# B&R Automation Studio project DiCoS_ACOPOStrak
Automation Studio 4.12.2.93; technology packages: mapp 5.21.0, mappCockpit 5.21.0, mappMotion 5.21.2, mappView 5.21.0

## Configuration Config2

CPU 5PC900.TS17-00, AutomationRuntime C4.90, Build 4.1.2, Safety 0.0, Vc V4.72.2

### Task classes (Cpu.sw)
```
Cyclic#1 (cycle 800 us, tolerance 0 us):
  trakFSM <- TrakControl.trakFSM.prg
  trakMove <- TrakControl.trakMove.prg
DataObjects: McAcpSys
Binaries: FWRules, McAcpSim, arcoal, arsvcreg, TCData, McAcpDrv, arflatprv, udbdef, McProfGen, mvLoader, mCoWebSc, asnxdb1, ConfAsmb, ConfSec, ConfShut, iomap, arconfig, asfw, ashwac, sysconf, User, Role, ashwd, Settings, Config_1, ConfPP, ConfCoup
Libraries: McBase, McAxis, McAcpTrak, AsIORTI, AsBrStr, McPureVAx, CoTrace, AsZip, FileIO, runtime, MpAxis, MpBase, McAcpAx, powerlnk, asieccon, arssl, asepl, MpData, sys_lib, DataObj, brsystem, astime
```

### Hardware
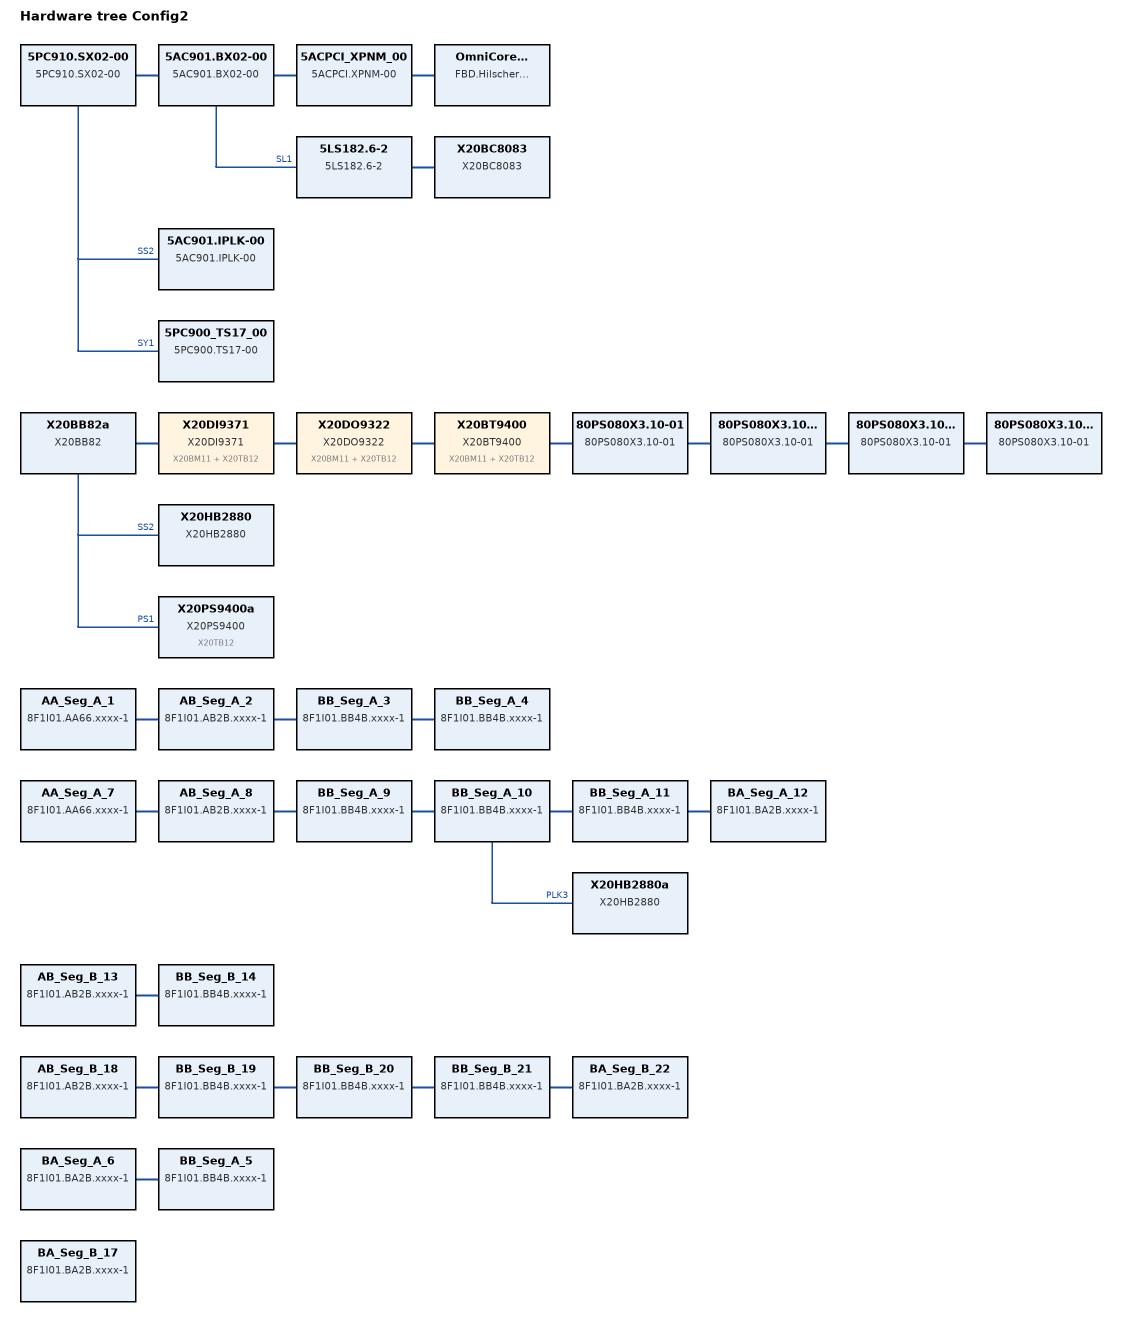
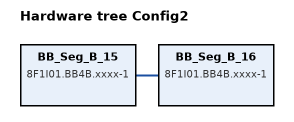
```
5AC901.BX02-00 : 5AC901.BX02-00 v1.0.1.0  [SY -> 5PC910.SX02-00.SY3]
5AC901.IPLK-00 : 5AC901.IPLK-00 v1.8.0.1  [SS -> 5PC910.SX02-00.SS2]
  Connector IF1:
    DNAConfiguration = manual
    EplNatSubnet = 192.168.102.0
5ACPCI_XPNM_00 : 5ACPCI.XPNM-00 v1.3.1.0  [SL -> 5AC901.BX02-00.SL2]
  Connector IF1:
    DtmId = d6364a6a-af48-4c58-9fae-63d24b23d839
  ConfigFile = 5ACPCI_XPNM_00.dtm
  ConfigModule = asnxdb1
5LS182.6-2 : 5LS182.6-2 v1.9.0.0  [SL -> 5AC901.BX02-00.SL1]
  Connector IF1:
    MtuSize = 1500
    CycleTime = 800
    EplNatSubnet = 192.168.103.0
5PC900_TS17_00 : 5PC900.TS17-00 v2.1.0.0  [SY -> 5PC910.SX02-00.SY1]
  ConfigurationID = APT_BFH_HW_Config
  TimerDeviceType = EPLX2X
  TimerDevice = 5LS182.6-2.IF1
  TaskClassIdleTime = 1600
  Cyclic1Duration = 800
  Cyclic1Tolerance = 0
  Cyclic3Duration = 49600
  Cyclic3Tolerance = 49600
  Cyclic8Duration = 9600
  FileDevice1
  FileDeviceName1 = SvgData
  FileDevicePath1 = C:\Users\nikla\Documents\BrAutomation\DiCoS_ACOPOStrak\Trak
  FileDevice2
  FileDeviceName2 = User
  FileDevicePath2 = C:\Users\nikla\Documents\BrAutomation\DiCoS_ACOPOStrak\Trak\User
  ActivateOpcUa = 1
  OpcUa_AuthenticationSecurityPolicy_EnableNone = 1
  OpcUa_AuthenticationSecurityPolicy_EnableBasic128Rsa15 = 1
  OpcUaInformationModels_PV_Version = 1
5PC910.SX02-00 : 5PC910.SX02-00 v2.1.0.0
  Connector IF1:
    AssignedOperatingSystem = ARemb
  Connector IF3:
    AssignedOperatingSystem = ARemb
    ActivateDevice = 1
    Mode = Manual
    InternetAddress = 192.168.1.220
    SubnetMask = 255.255.255.0
  Connector IF4:
    AssignedOperatingSystem = ARemb
    ActivateDevice = 1
    Mode = Manual
    InternetAddress = 10.0.0.3
    SubnetMask = 255.255.255.0
    ActivateSnmp = 2
  Connector IF5:
    AssignedOperatingSystem = ARemb
  Connector IF6:
    AssignedOperatingSystem = ARemb
  Connector IF7:
    AssignedOperatingSystem = ARemb
  Connector IF8:
    AssignedOperatingSystem = ARemb
  Connector IF9:
    AssignedOperatingSystem = ARemb
80PS080X3.10-01 : 80PS080X3.10-01 v1.5.0.0  [X2X1 -> X20BT9400.X2X1 [Cable Type=X2XCable, Length=10, Version=1.0.0.3]]
  Supervision = off
  ParallelMode01 = on
  VoltageSet01 = 58
  RampMode01 = steep
  ChopperEnable01 = on
80PS080X3.10-01a : 80PS080X3.10-01 v1.5.0.0  [X2X1 -> 80PS080X3.10-01.X2X2 [Cable Type=X2XCable, Length=10, Version=1.0.0.3]]
  Supervision = off
  ParallelMode01 = on
  VoltageSet01 = 58
  RampMode01 = steep
  ChopperEnable01 = on
80PS080X3.10-01b : 80PS080X3.10-01 v1.5.0.0  [X2X1 -> 80PS080X3.10-01a.X2X2 [Cable Type=X2XCable, Length=10, Version=1.0.0.3]]
  Supervision = off
  ParallelMode01 = on
  VoltageSet01 = 58
  RampMode01 = steep
  ChopperEnable01 = on
80PS080X3.10-01c : 80PS080X3.10-01 v1.5.0.0  [X2X1 -> 80PS080X3.10-01b.X2X2 [Cable Type=X2XCable, Length=10, Version=1.0.0.3]]
  Supervision = off
  ParallelMode01 = on
  VoltageSet01 = 58
  RampMode01 = steep
  ChopperEnable01 = on
AA_Seg_A_1 : 8F1I01.AA66.xxxx-1 v1.0.0.2  [PLK1 -> BA_Seg_A_12.PLK2 (NodeNumber=1) [Cable Type=PowerlinkCable, Length=10, Version=1.0.0.3]; PLK2 -> AB_Seg_A_2.PLK1 (NodeNumber=1) [Cable Type=PowerlinkCable, Length=10, Version=1.0.0.3]]
  EnableDNA = on
  DriveConfiguration:
    McTypeID = LLMConfig
  DriveConfiguration/Segment:
    Shape = STRAIGHT660
    SegmentReference = Seg_A_1
    StopReaction = UseAssemblySetting
    SpeedFilter = UseAssemblySetting
AA_Seg_A_7 : 8F1I01.AA66.xxxx-1 v1.0.0.2  [PLK1 -> BA_Seg_A_6.PLK2 (NodeNumber=7) [Cable Type=PowerlinkCable, Length=10, Version=1.0.0.3]; PLK2 -> AB_Seg_A_8.PLK1 (NodeNumber=7) [Cable Type=PowerlinkCable, Length=10, Version=1.0.0.3]]
  EnableDNA = on
  DriveConfiguration:
    McTypeID = LLMConfig
  DriveConfiguration/Segment:
    Shape = STRAIGHT660
    SegmentReference = Seg_A_7
    SegmentSectorDirection = Positive
    ElongationCompensation = UseAssemblySetting
    StopReaction = UseAssemblySetting
    SpeedFilter = UseAssemblySetting
AB_Seg_A_2 : 8F1I01.AB2B.xxxx-1 v1.0.0.2  [PLK1 -> AA_Seg_A_1.PLK2 (NodeNumber=2) [Cable Type=PowerlinkCable, Length=10, Version=1.0.0.3]; PLK2 -> BB_Seg_A_3.PLK1 (NodeNumber=2) [Cable Type=PowerlinkCable, Length=10, Version=1.0.0.3]]
  EnableDNA = on
  DriveConfiguration:
    McTypeID = LLMConfig
  DriveConfiguration/Segment:
    Shape = STRAIGHT105_TO_CIRCULAR
    SegmentReference = Seg_A_2
    StopReaction = UseAssemblySetting
    SpeedFilter = UseAssemblySetting
AB_Seg_A_8 : 8F1I01.AB2B.xxxx-1 v1.0.0.2  [PLK1 -> AA_Seg_A_7.PLK2 (NodeNumber=8) [Cable Type=PowerlinkCable, Length=10, Version=1.0.0.3]; PLK2 -> BB_Seg_A_9.PLK1 (NodeNumber=8) [Cable Type=PowerlinkCable, Length=10, Version=1.0.0.3]]
  EnableDNA = on
  DriveConfiguration:
    McTypeID = LLMConfig
  DriveConfiguration/Segment:
    Shape = STRAIGHT105_TO_CIRCULAR
    SegmentReference = Seg_A_8
    StopReaction = UseAssemblySetting
    SpeedFilter = UseAssemblySetting
AB_Seg_B_13 : 8F1I01.AB2B.xxxx-1 v1.0.0.2  [PLK1 -> BA_Seg_B_22.PLK2 (NodeNumber=13) [Cable Type=PowerlinkCable, Length=10, Version=1.0.0.3]; PLK2 -> BB_Seg_B_14.PLK1 (NodeNumber=13) [Cable Type=PowerlinkCable, Length=10, Version=1.0.0.3]]
  EnableDNA = on
  DriveConfiguration:
    McTypeID = LLMConfig
  DriveConfiguration/Segment:
    Shape = STRAIGHT105_TO_CIRCULAR
    SegmentReference = Seg_B_13
    StopReaction = UseAssemblySetting
    SpeedFilter = UseAssemblySetting
AB_Seg_B_18 : 8F1I01.AB2B.xxxx-1 v1.0.0.2  [PLK1 -> BA_Seg_B_17.PLK2 (NodeNumber=18) [Cable Type=PowerlinkCable, Length=10, Version=1.0.0.3]; PLK2 -> BB_Seg_B_19.PLK1 (NodeNumber=18) [Cable Type=PowerlinkCable, Length=10, Version=1.0.0.3]]
  EnableDNA = on
  DriveConfiguration:
    McTypeID = LLMConfig
  DriveConfiguration/Segment:
    Shape = STRAIGHT105_TO_CIRCULAR
    SegmentReference = Seg_B_18
    StopReaction = UseAssemblySetting
    SpeedFilter = UseAssemblySetting
BA_Seg_A_12 : 8F1I01.BA2B.xxxx-1 v1.0.0.2  [PLK1 -> BB_Seg_A_11.PLK2 (NodeNumber=12) [Cable Type=PowerlinkCable, Length=10, Version=1.0.0.3]; PLK2 -> AA_Seg_A_1.PLK1 (NodeNumber=12) [Cable Type=PowerlinkCable, Length=10, Version=1.0.0.3]]
  EnableDNA = on
  DriveConfiguration:
    McTypeID = LLMConfig
  DriveConfiguration/Segment:
    Shape = CIRCULAR_TO_STRAIGHT105
    SegmentReference = Seg_A_12
    StopReaction = UseAssemblySetting
    SpeedFilter = UseAssemblySetting
BA_Seg_A_6 : 8F1I01.BA2B.xxxx-1 v1.0.0.2  [PLK1 -> BB_Seg_A_5.PLK2 (NodeNumber=6) [Cable Type=PowerlinkCable, Length=10, Version=1.0.0.3]; PLK2 -> AA_Seg_A_7.PLK1 (NodeNumber=6) [Cable Type=PowerlinkCable, Length=10, Version=1.0.0.3]]
  EnableDNA = on
  DriveConfiguration:
    McTypeID = LLMConfig
  DriveConfiguration/Segment:
    Shape = CIRCULAR_TO_STRAIGHT105
    SegmentReference = Seg_A_6
    StopReaction = UseAssemblySetting
    SpeedFilter = UseAssemblySetting
BA_Seg_B_17 : 8F1I01.BA2B.xxxx-1 v1.0.0.2  [PLK1 -> BB_Seg_B_16.PLK2 (NodeNumber=17) [Cable Type=PowerlinkCable, Length=10, Version=1.0.0.3]; PLK2 -> AB_Seg_B_18.PLK1 (NodeNumber=17) [Cable Type=PowerlinkCable, Length=10, Version=1.0.0.3]]
  EnableDNA = on
  DriveConfiguration:
    McTypeID = LLMConfig
  DriveConfiguration/Segment:
    Shape = CIRCULAR_TO_STRAIGHT105
    SegmentReference = Seg_B_17
    StopReaction = UseAssemblySetting
    SpeedFilter = UseAssemblySetting
BA_Seg_B_22 : 8F1I01.BA2B.xxxx-1 v1.0.0.2  [PLK1 -> BB_Seg_B_21.PLK2 (NodeNumber=22) [Cable Type=PowerlinkCable, Length=10, Version=1.0.0.3]; PLK2 -> AB_Seg_B_13.PLK1 (NodeNumber=22) [Cable Type=PowerlinkCable, Length=10, Version=1.0.0.3]]
  EnableDNA = on
  DriveConfiguration:
    McTypeID = LLMConfig
  DriveConfiguration/Segment:
    Shape = CIRCULAR_TO_STRAIGHT105
    SegmentReference = Seg_B_22
    StopReaction = UseAssemblySetting
    SpeedFilter = UseAssemblySetting
BB_Seg_A_10 : 8F1I01.BB4B.xxxx-1 v1.0.0.2  [PLK1 -> BB_Seg_A_9.PLK2 (NodeNumber=10) [Cable Type=PowerlinkCable, Length=10, Version=1.0.0.3]; PLK2 -> BB_Seg_A_11.PLK1 (NodeNumber=10) [Cable Type=PowerlinkCable, Length=10, Version=1.0.0.3]; PLK3 -> X20HB2880a.ETH1 (NodeNumber=10) [Cable Type=PowerlinkCable, Length=10, Version=1.0.0.3]]
  EnableDNA = on
  DriveConfiguration:
    McTypeID = LLMConfig
  DriveConfiguration/Segment:
    Shape = CIRCULAR
    SegmentReference = Seg_A_10
    StopReaction = UseAssemblySetting
    SpeedFilter = UseAssemblySetting
BB_Seg_A_11 : 8F1I01.BB4B.xxxx-1 v1.0.0.2  [PLK1 -> BB_Seg_A_10.PLK2 (NodeNumber=11) [Cable Type=PowerlinkCable, Length=10, Version=1.0.0.3]; PLK2 -> BA_Seg_A_12.PLK1 (NodeNumber=11) [Cable Type=PowerlinkCable, Length=10, Version=1.0.0.3]]
  EnableDNA = on
  DriveConfiguration:
    McTypeID = LLMConfig
  DriveConfiguration/Segment:
    Shape = CIRCULAR
    SegmentReference = Seg_A_11
    StopReaction = UseAssemblySetting
    SpeedFilter = UseAssemblySetting
BB_Seg_A_3 : 8F1I01.BB4B.xxxx-1 v1.0.0.2  [PLK1 -> AB_Seg_A_2.PLK2 (NodeNumber=3) [Cable Type=PowerlinkCable, Length=10, Version=1.0.0.3]; PLK2 -> BB_Seg_A_4.PLK1 (NodeNumber=3) [Cable Type=PowerlinkCable, Length=10, Version=1.0.0.3]]
  EnableDNA = on
  DriveConfiguration:
    McTypeID = LLMConfig
  DriveConfiguration/Segment:
    Shape = CIRCULAR
    SegmentReference = Seg_A_3
    StopReaction = UseAssemblySetting
    SpeedFilter = UseAssemblySetting
BB_Seg_A_4 : 8F1I01.BB4B.xxxx-1 v1.0.0.2  [PLK1 -> BB_Seg_A_3.PLK2 (NodeNumber=4) [Cable Type=PowerlinkCable, Length=10, Version=1.0.0.3]]
  EnableDNA = on
  DriveConfiguration:
    McTypeID = LLMConfig
  DriveConfiguration/Segment:
    Shape = CIRCULAR
    SegmentReference = Seg_A_4
    StopReaction = UseAssemblySetting
    SpeedFilter = UseAssemblySetting
BB_Seg_A_5 : 8F1I01.BB4B.xxxx-1 v1.0.0.2  [PLK2 -> BA_Seg_A_6.PLK1 (NodeNumber=5) [Cable Type=PowerlinkCable, Length=10, Version=1.0.0.3]]
  EnableDNA = on
  DriveConfiguration:
    McTypeID = LLMConfig
  DriveConfiguration/Segment:
    Shape = CIRCULAR
    SegmentReference = Seg_A_5
    StopReaction = UseAssemblySetting
    SpeedFilter = UseAssemblySetting
BB_Seg_A_9 : 8F1I01.BB4B.xxxx-1 v1.0.0.2  [PLK1 -> AB_Seg_A_8.PLK2 (NodeNumber=9) [Cable Type=PowerlinkCable, Length=10, Version=1.0.0.3]; PLK2 -> BB_Seg_A_10.PLK1 (NodeNumber=9) [Cable Type=PowerlinkCable, Length=10, Version=1.0.0.3]]
  EnableDNA = on
  DriveConfiguration:
    McTypeID = LLMConfig
  DriveConfiguration/Segment:
    Shape = CIRCULAR
    SegmentReference = Seg_A_9
    StopReaction = UseAssemblySetting
    SpeedFilter = UseAssemblySetting
BB_Seg_B_14 : 8F1I01.BB4B.xxxx-1 v1.0.0.2  [PLK1 -> AB_Seg_B_13.PLK2 (NodeNumber=14) [Cable Type=PowerlinkCable, Length=10, Version=1.0.0.3]]
  EnableDNA = on
  DriveConfiguration:
    McTypeID = LLMConfig
  DriveConfiguration/Segment:
    Shape = CIRCULAR
    SegmentReference = Seg_B_14
    StopReaction = UseAssemblySetting
    SpeedFilter = UseAssemblySetting
BB_Seg_B_15 : 8F1I01.BB4B.xxxx-1 v1.0.0.2  [PLK2 -> BB_Seg_B_16.PLK1 (NodeNumber=15) [Cable Type=PowerlinkCable, Length=10, Version=1.0.0.3]]
  EnableDNA = on
  DriveConfiguration:
    McTypeID = LLMConfig
  DriveConfiguration/Segment:
    Shape = CIRCULAR
    SegmentReference = Seg_B_15
    StopReaction = UseAssemblySetting
    SpeedFilter = UseAssemblySetting
BB_Seg_B_16 : 8F1I01.BB4B.xxxx-1 v1.0.0.2  [PLK1 -> BB_Seg_B_15.PLK2 (NodeNumber=16) [Cable Type=PowerlinkCable, Length=10, Version=1.0.0.3]; PLK2 -> BA_Seg_B_17.PLK1 (NodeNumber=16) [Cable Type=PowerlinkCable, Length=10, Version=1.0.0.3]]
  EnableDNA = on
  DriveConfiguration:
    McTypeID = LLMConfig
  DriveConfiguration/Segment:
    Shape = CIRCULAR
    SegmentReference = Seg_B_16
    StopReaction = UseAssemblySetting
    SpeedFilter = UseAssemblySetting
BB_Seg_B_19 : 8F1I01.BB4B.xxxx-1 v1.0.0.2  [PLK1 -> AB_Seg_B_18.PLK2 (NodeNumber=19) [Cable Type=PowerlinkCable, Length=10, Version=1.0.0.3]; PLK2 -> BB_Seg_B_20.PLK1 (NodeNumber=19) [Cable Type=PowerlinkCable, Length=10, Version=1.0.0.3]]
  EnableDNA = on
  DriveConfiguration:
    McTypeID = LLMConfig
  DriveConfiguration/Segment:
    Shape = CIRCULAR
    SegmentReference = Seg_B_19
    StopReaction = UseAssemblySetting
    SpeedFilter = UseAssemblySetting
BB_Seg_B_20 : 8F1I01.BB4B.xxxx-1 v1.0.0.2  [PLK1 -> BB_Seg_B_19.PLK2 (NodeNumber=20) [Cable Type=PowerlinkCable, Length=10, Version=1.0.0.3]; PLK2 -> BB_Seg_B_21.PLK1 (NodeNumber=20) [Cable Type=PowerlinkCable, Length=10, Version=1.0.0.3]; PLK3 -> X20HB2880a.ETH2 (NodeNumber=20) [Cable Type=PowerlinkCable, Length=10, Version=1.0.0.3]]
  EnableDNA = on
  DriveConfiguration:
    McTypeID = LLMConfig
  DriveConfiguration/Segment:
    Shape = CIRCULAR
    SegmentReference = Seg_B_20
    StopReaction = UseAssemblySetting
    SpeedFilter = UseAssemblySetting
BB_Seg_B_21 : 8F1I01.BB4B.xxxx-1 v1.0.0.2  [PLK1 -> BB_Seg_B_20.PLK2 (NodeNumber=21) [Cable Type=PowerlinkCable, Length=10, Version=1.0.0.3]; PLK2 -> BA_Seg_B_22.PLK1 (NodeNumber=21) [Cable Type=PowerlinkCable, Length=10, Version=1.0.0.3]]
  EnableDNA = on
  DriveConfiguration:
    McTypeID = LLMConfig
  DriveConfiguration/Segment:
    Shape = CIRCULAR
    SegmentReference = Seg_B_21
    StopReaction = UseAssemblySetting
    SpeedFilter = UseAssemblySetting
OmniCore_Standard : FBD.Hilscher.PNIOGenDevDTM2.OmniCore Standard v1.1 (OrderNumber=OmniCore Standard, VendorAddress=omnicore)  [PN1 -> 5ACPCI_XPNM_00.IF1]
  DtmId = 5f4a343d-d0a2-4fff-bfd8-5abcfec9ae3d
X20BB82a : X20BB82 v1.1.0.0
  Connector IF1:
    CycleTime = 1600
X20BC8083 : X20BC8083 v2.14.0.0  [PLK1 -> 5LS182.6-2.IF1 (NodeNumber=23) [Cable Type=PowerlinkCable, Length=10, Version=1.0.0.3]; SL -> X20BB82a.SL1]
  Supervision = off
  EPL_Chained = on
  EnableDNA = on
X20BM11 : X20BM11 v1.1.0.0  [X2X1 -> X20BM11b.X2X2]
X20BM11a : X20BM11 v1.1.0.0  [X2X1 -> X20BB82a.IF1]
X20BM11b : X20BM11 v1.1.0.0  [X2X1 -> X20BM11a.X2X2]
X20BT9400 : X20BT9400 v1.3.0.0  [SS1 -> X20TB12.SS; SL -> X20BM11.SL1]
  Supervision = off
X20DI9371 : X20DI9371 v1.4.0.0  [SS1 -> X20TB12b.SS; SL -> X20BM11a.SL1]
X20DO9322 : X20DO9322 v1.5.0.0  [SS1 -> X20TB12c.SS; SL -> X20BM11b.SL1]
X20HB2880 : X20HB2880 v1.2.0.0  [SS -> X20BB82a.SS2]
X20HB2880a : X20HB2880 v1.2.0.0  [ETH1 -> BB_Seg_A_10.PLK3 [Cable Type=PowerlinkCable, Length=10, Version=1.0.0.3]; ETH2 -> BB_Seg_B_20.PLK3 [Cable Type=PowerlinkCable, Length=10, Version=1.0.0.3]; SS -> X20BB82a.SS1]
X20PS9400a : X20PS9400 v1.8.0.0  [SS1 -> X20TB12a.SS; PS -> X20BB82a.PS1]
X20TB12 : X20TB12 v1.0.0.0
X20TB12a : X20TB12 v1.0.0.0
X20TB12b : X20TB12 v1.0.0.0
X20TB12c : X20TB12 v1.0.0.0
```

### ConfAsmb.assembly - 5PC900_TS17_00/mappMotion/ConfAsmb.assembly
```
Element gAssemblyFigure8 (Type=assembly)
  Tracks:
    TrackSeparation = 0.030
    Track[1]:
      Segments:
        SegmentRef[1] = ::Seg_A_1
        SegmentRef[2] = ::Seg_A_2
        SegmentRef[3] = ::Seg_A_3
        SegmentRef[4] = ::Seg_A_4
        SegmentRef[5] = ::Seg_A_5
        SegmentRef[6] = ::Seg_A_6
        SegmentRef[7] = ::Seg_A_7
        SegmentRef[8] = ::Seg_A_8
        SegmentRef[9] = ::Seg_A_9
        SegmentRef[10] = ::Seg_A_10
        SegmentRef[11] = ::Seg_A_11
        SegmentRef[12] = ::Seg_A_12
      Position = Absolute
        SegmentRef = ::Seg_A_1
        SegmentCountDirection = RightToLeft
        Translation:
          X = 0.0
          Y = 0.0
          Z = 0.0
        Orientation:
          Angle1 = 0.0
          Angle2 = 0.0
          Angle3 = 180.0
    Track[2]:
      Segments:
        SegmentRef[1] = ::Seg_B_13
        SegmentRef[2] = ::Seg_B_14
        SegmentRef[3] = ::Seg_B_15
        SegmentRef[4] = ::Seg_B_16
        SegmentRef[5] = ::Seg_B_17
        SegmentRef[6] = ::Seg_B_18
        SegmentRef[7] = ::Seg_B_19
        SegmentRef[8] = ::Seg_B_20
        SegmentRef[9] = ::Seg_B_21
        SegmentRef[10] = ::Seg_B_22
      Position = RelativeToOne
        TrackSegmentPosition:
          SegmentRef = ::Seg_B_13
        Base:
          SegmentRef = ::Seg_A_7
          Position = 0.329907
  CommonSegmentSettings:
    SegmentSimulationOnPLC = Off
    ElongationCompensation = Inactive
    StopReaction = InductionHalt
    SpeedFilter = Lowpass
      FilterTime = 0.0008
    ControllerParameters:
      DefaultParameter:
        Controller:
          Position:
            ProportionalGain = 150
          Speed:
            ProportionalGain = 80
            IntegrationTime = 0
          FeedForward:
            TotalMass = 0.7
            ForcePositive = 1.5
            ForceNegative = 1.5
            SpeedForceFactor = 1.4
            ForceLoad = 0.0
        MovementErrorLimits:
          PositionError = 0.03
          VelocityError = 50
      AdditionalParameterSets = NotUsed
    ScopeOfErrorReaction = Assembly
    ShuttleIdentificationTime = 0
  Shuttles:
    MaxShuttleCount = 10
    MaxShuttleCommandCount = 0
    UseConvoys = Active
    DistanceReserve:
      Collision = 0.002
      ErrorStop = 0.006
    ShuttleStereotypes:
      ShuttleStRef[1] = gShuttleStereotype_1
    MagnetPlateConfigurations:
      ShuttleType[1] = 8F1SA.100.xxxxxx-x
    CollisionAvoidance:
      Strategy = Constant
      MaximumModelDimensions:
        Length:
          ExtentToFront = 0.046
          ExtentToBack = 0.046
        Width:
          Width = 0.046
  AssemblyFeatures:
    AssemblyFeatureRef[1] = Feature_Coupling
  Visualization:
    MonitoringPv = ::trakAsmb.monData
    ProcessingTaskClass = 1
```

### ConfCoup.assemblyfeature - 5PC900_TS17_00/mappMotion/ConfCoup.assemblyfeature
```
Element Feature_Coupling (Type=assemblyfeature)
  Type = Coupling
    CouplingObject[1]:
      Name = couplingLoad
      ShuttleCount = 1
      CamAutomat
      CamList
```

### ConfPP.processpointlist - 5PC900_TS17_00/mappMotion/ConfPP.processpointlist
```
Element gPPList (Type=processpointlist)
  ProcessPoint[0]:
    Name = gPPDepot
    SectorRef = gSecFull
    Position = 5.6
    TriggerEventBufferSize = 10
    BarrierFunctionality = On
```

### ConfSec.sector - 5PC900_TS17_00/mappMotion/ConfSec.sector
```
Element gSecMajor (Type=sector)
  Type = Composed
    StartSegment:
      SegmentRef = ::Seg_A_3
    IntermediateSegments:
      SegmentRef[1] = ::Seg_A_2
      SegmentRef[2] = ::Seg_A_1
      SegmentRef[3] = ::Seg_A_12
      SegmentRef[4] = ::Seg_A_11
      SegmentRef[5] = ::Seg_A_10
      SegmentRef[6] = ::Seg_A_9
      SegmentRef[7] = ::Seg_A_8
      SegmentRef[8] = ::Seg_A_7
      SegmentRef[9] = ::Seg_A_6
      SegmentRef[10] = ::Seg_A_5
    EndSegment:
      SegmentRef = ::Seg_A_4
      PositionRelativeTo = FromEnd
Element gSecMinor (Type=sector)
  Type = Composed
    StartSegment:
      SegmentRef = ::Seg_B_18
    IntermediateSegments:
      SegmentRef[1] = ::Seg_B_19
      SegmentRef[2] = ::Seg_B_20
      SegmentRef[3] = ::Seg_B_21
      SegmentRef[4] = ::Seg_B_22
      SegmentRef[5] = ::Seg_B_13
      SegmentRef[6] = ::Seg_B_14
      SegmentRef[7] = ::Seg_B_15
      SegmentRef[8] = ::Seg_B_16
    EndSegment:
      SegmentRef = ::Seg_B_17
      PositionRelativeTo = FromEnd
Element gSecLoad (Type=sector)
  Type = Subsector
    SectorRef = gSecMajor
    Start:
      Position = 0.3
    Length = 0.6
    Direction = Positive
Element gSecFull (Type=sector)
  Type = Composed
    StartSegment:
      SegmentRef = ::Seg_A_5
      PositionRelativeTo = FromEnd
    IntermediateSegments:
      SegmentRef[1] = ::Seg_A_4
      SegmentRef[2] = ::Seg_A_3
      SegmentRef[3] = ::Seg_A_2
      SegmentRef[4] = ::Seg_A_1
      SegmentRef[5] = ::Seg_A_12
      SegmentRef[6] = ::Seg_A_11
      SegmentRef[7] = ::Seg_A_10
      SegmentRef[8] = ::Seg_A_9
      SegmentRef[9] = ::Seg_A_8
      SegmentRef[10] = ::Seg_A_7
      SegmentRef[11] = ::Seg_B_13
      SegmentRef[12] = ::Seg_B_14
      SegmentRef[13] = ::Seg_B_15
      SegmentRef[14] = ::Seg_B_16
      SegmentRef[15] = ::Seg_B_17
      SegmentRef[16] = ::Seg_B_18
      SegmentRef[17] = ::Seg_B_19
      SegmentRef[18] = ::Seg_B_20
      SegmentRef[19] = ::Seg_B_21
      SegmentRef[20] = ::Seg_B_22
      SegmentRef[21] = ::Seg_A_7
    EndSegment:
      SegmentRef = ::Seg_A_6
```

### ConfShut.shuttlestereotype - 5PC900_TS17_00/mappMotion/ConfShut.shuttlestereotype
```
Element gShuttleStereotype_1 (Type=shuttlestereotype)
  MeasurementUnit = 5067858
  MeasurementResolution = 0.00001
  MovementLimits = Internal
    VelocityIsReadOnly = 0
    Velocity:
      Velocity = 4
    AccelerationIsReadOnly = 0
    Acceleration:
      Acceleration = 40
    DecelerationIsReadOnly = 0
    Deceleration:
      Deceleration = 40
  JerkFilter = Used
    JerkTime = 0.02
  UserData:
    Size = 0
```

### Config_1.axis - 5PC900_TS17_00/mappMotion/Config_1.axis
```
Element gDummyAxis (Type=axis)
  BaseTypeIsReadOnly = 0
  BaseType = LinearBounded
    MeasurementUnit = 5066068
    MeasurementResolutionIsReadOnly = 0
    MeasurementResolution = 0.01
    CountDirectionIsReadOnly = 0
    CountDirection = Standard
  MovementLimitsIsReadOnly = 0
  MovementLimits = Internal
    Position:
      LowerLimitMin = -1.79769313486231E308
      UpperLimitMax = 1.79769313486231E308
      LowerLimit = -1000.0
      UpperLimit = 1000.0
    VelocityIsReadOnly = 0
    Velocity:
      VelocityMax = 3.4E38
      Velocity = 10.0
    AccelerationIsReadOnly = 0
    Acceleration:
      AccelerationMax = 3.4E38
      Acceleration = 50.0
    DecelerationIsReadOnly = 0
    Deceleration:
      DecelerationMax = 3.4E38
      Deceleration = 50.0
  Alarms = None
```

## Logical view

Binary libraries used (declarations not repeated): operator, runtime, astime, AsIecCon, AsIORTI, AsBrStr, AsZip, FileIO, sys_lib, DataObj, brsystem, McBase, MpAxis 5.21.2, McPureVAx 5.21.2, McAcpAx 5.21.2, McAcpTrak, McAxis, MpBase, MpData 5.21.0, CoTrace

### Global.typ - Globale Datentypen
```iecst
(*OPC UA Interface*)

TYPE
	trakMes_t : 	STRUCT
		cmd : trakMesCmd_t; (*Kommandos MES -> trak*)
		state : trakMesState_t; (*Status trak -> MES*)
	END_STRUCT;
	trakMesCmd_t : 	STRUCT
		goABB : BOOL; (*Setzen durch MES, Rücksetzen durch trak FSM als Kommando Bestätigung*)
		goDelta : BOOL; (*Setzen durch MES, Rücksetzen durch trak FSM als Kommando Bestätigung*)
	END_STRUCT;
	trakMesState_t : 	STRUCT
		power : BOOL; (*trak Assembly ist On*)
		atABB : BOOL; (*Shuttle beim ABB Roboter*)
		atDelta : BOOL; (*Shuttle beim Delta Roboter*)
	END_STRUCT;
END_TYPE

(*Assembly Interface*)

TYPE
	trakState_t : 	STRUCT
		ready : BOOL;
		loading : BOOL; (*Führe Get-Shuttle FSM aus, Assembly bereit aber Shuttle Referenzen noch nicht*)
		homing : BOOL;
		stopping : BOOL;
		disabled : BOOL;
		errorStop : BOOL;
	END_STRUCT;
	trakAsmbCmd_t : 	STRUCT
		simulation : USINT; (*Wenn >0, dann ist Simulationsmodus aktiv bez. diese Anzahl an Shuttles wird simuliert*)
		reload : BOOL; (*Neuladen aller Shuttles*)
		reset : {REDUND_UNREPLICABLE} BOOL; (*Beim setzen auf 1 wird Asmb zurückgesetzt.*)
		power : BOOL; (*Beim setzen auf 1 wird automatisch Asmb FSM bis auf Zustand Ready gebracht.*)
	END_STRUCT;
	trakShuttle_t : 	STRUCT
		id : UINT;
		axis : McAxisType;
	END_STRUCT;
	trakAsmb_t : 	STRUCT
		monData : McAcpTrakAssemblyMonData;
		shuttleCount : UINT; (*Anzahl gefundener Shuttles*)
		shuttles : ARRAY[0..9]OF trakShuttle_t; (*Referenzen auf Shuttle Achsen & IDs*)
		state : trakState_t;
		cmd : trakAsmbCmd_t;
	END_STRUCT;
	New_Datatype : 	STRUCT
	END_STRUCT;
END_TYPE

(*Single Interface*)

TYPE
	trakSingleCmd_t : 	STRUCT
		goABB : BOOL;
		goDelta : BOOL;
		read : BOOL;
	END_STRUCT;
	trakSingleState_t : 	STRUCT
		moving : BOOL;
		atABB : BOOL;
		atDelta : BOOL;
	END_STRUCT;
	trakSingle_t : 	STRUCT
		cmd : trakSingleCmd_t;
		state : trakSingleState_t;
	END_STRUCT;
END_TYPE

(*Convoy Interface*)

TYPE
	trakConvoyCmd_t : 	STRUCT
		reset : BOOL;
		prepare : BOOL;
		couple : BOOL;
		move : BOOL;
		release : BOOL;
		return : BOOL;
	END_STRUCT;
	trakConvoyState_t : 	STRUCT
		prepared : BOOL;
		coupled : BOOL;
		moved : BOOL;
		released : BOOL;
		returned : BOOL;
	END_STRUCT;
	trakConvoy_t : 	STRUCT
		state : trakConvoyState_t;
		cmd : trakConvoyCmd_t;
		startPos : LREAL;
		coupleDistance : LREAL;
		targetPos : LREAL;
	END_STRUCT;
END_TYPE
```

### Global.var - Globale Variablen
```iecst
(*OPC UA Interface*)
VAR
	trakMES : trakMes_t;
END_VAR
(*Assembly Interface*)
VAR
	trakAsmb : trakAsmb_t;
END_VAR
(*Single Interface*)
VAR
	trakSingle : trakSingle_t;
END_VAR
(*Convoy Interface*)
VAR
	trakConvoy : trakConvoy_t;
END_VAR
```


### Program Logical/TrakControl/trakAsmb (IEC)

#### Variables.var
```iecst
(*Interne FBs*)
VAR
	FB_status : MC_BR_AsmReadStatus_AcpTrak;
	FB_reset : MC_BR_AsmReset_AcpTrak;
	FB_powerOff : MC_BR_AsmPowerOff_AcpTrak;
	FB_powerOn : MC_BR_AsmPowerOn_AcpTrak;
	FB_getShuttle : MC_BR_AsmGetShuttle_AcpTrak;
	FB_addShuttle : MC_BR_SecAddShuttle_AcpTrak;
END_VAR
(*Interne Variablen*)
VAR
	simShuttleCount : USINT;
	getShuttleStep : intGetShuttleStep_t;
END_VAR
```

#### Main.st
```iecst
PROGRAM _INIT
	// Initialsiere alle FBs
	FB_status.Assembly := ADR(gAssemblyFigure8);
	FB_reset.Assembly := ADR(gAssemblyFigure8);
	FB_powerOff.Assembly := ADR(gAssemblyFigure8);
	FB_powerOn.Assembly := ADR(gAssemblyFigure8);
	FB_getShuttle.Assembly := ADR(gAssemblyFigure8);
	FB_addShuttle.Sector := ADR(gSecMinor);
	FB_addShuttle.Sector := ADR(gSecMajor);
	FB_addShuttle.Sector := ADR(gSecFull);

	// alle FBs ausser status deaktivieren
	FB_reset.Execute := FALSE;
	FB_powerOff.Execute := FALSE;
	FB_powerOn.Execute := FALSE;
	FB_getShuttle.Enable := FALSE;

	// Status FB aktivieren
	FB_status.Enable := TRUE;

	// Shuttle-Get FSM auf Reset
	getShuttleStep := getShuttleRESET;
	simShuttleCount := 0;

	// Initiale Kommandos
	trakAsmb.cmd.simulation := 0;
	trakAsmb.cmd.reload := FALSE;
	trakAsmb.cmd.reset := FALSE;
	trakAsmb.cmd.power := FALSE;

END_PROGRAM

PROGRAM _CYCLIC
	// Was ist der Zustand des Assembly?
	trakAsmb.state.errorStop := FB_status.AssemblyErrorStop;
	trakAsmb.state.disabled := FB_status.AssemblyDisabled;
	trakAsmb.state.homing := FB_status.AssemblyHoming;
	trakAsmb.state.stopping := FB_status.AssemblyStopping;
	// Wir sind die Shuttles am laden wenn Assembly bereit, aber Shuttle-Get FSM noch nicht.
	trakAsmb.state.loading := FB_status.AssemblyReady AND (getShuttleStep <> getShuttleDONE) AND getShuttleStep > getShuttleWAIT;
	// Wir sind komplett Bereit wenn Assembly und Shuttle-Get FSM bereit.
	trakAsmb.state.ready := FB_status.AssemblyReady AND getShuttleStep = getShuttleDONE;

	// Einschaltbefehl zurücksetzen wenn Zustand Ready verlassen wird.
	IF EDGENEG(FB_status.AssemblyReady) THEN
		trakAsmb.cmd.power := FALSE;
	END_IF;

	// Sind wir im Error oder wollen wir manuell Zurücksetzen? => Assembly zurücksetzen
	IF trakAsmb.state.errorStop OR trakAsmb.cmd.reset THEN
		FB_reset.Execute := TRUE;
		getShuttleStep := getShuttleRESET;
		trakAsmb.cmd.power := FALSE;
	END_IF;

	// Nach Reset kommen wir in Disabled, mit Einschaltbefehl ein PowerOn durchführen.
	IF trakAsmb.state.disabled AND trakAsmb.cmd.power THEN
		FB_powerOn.Execute := TRUE;
	END_IF;

	// Sind wir in Homing/Loading/Ready aber ohne Einschaltbefehl? => Stoppe Assembly
	IF (trakAsmb.state.homing OR trakAsmb.state.loading OR trakAsmb.state.ready) AND NOT trakAsmb.cmd.power THEN
		FB_powerOff.Execute := TRUE;
	END_IF;

	// Befehl zum Neuladen der Shuttles erhalten? => Get-Shuttle FSM zurücksetzen.
	IF (trakAsmb.cmd.reload AND getShuttleStep = getShuttleDONE) THEN
		getShuttleStep := getShuttleRESET;
		trakAsmb.cmd.reload := FALSE;
	END_IF;

	// Durchlaufe eine FSM um die Shuttlereferenzen per getShuttle FB zu erhalten.
	CASE getShuttleStep OF
		getShuttleRESET:
			// lösche die komplette Referenzstruktur
			brsmemset(ADR(trakAsmb.shuttles), 0, SIZEOF(trakAsmb.shuttles));
			//trakAsmb.shuttleCount := 0;
			// warte auf nächsten Wechsel in Ready
			getShuttleStep := getShuttleWAIT;

		getShuttleWAIT:
			// Warte bis Assembly in Zustand Ready übergeht.
			IF FB_status.AssemblyReady THEN
				// wenn die Anzahl Simulierte Shuttles noch nicht erreicht
				//  > dann Virtuelle hinzufügen
				//  > ansonsten nur die echten laden
				IF trakAsmb.cmd.simulation <> 0 AND trakAsmb.cmd.simulation <> trakAsmb.shuttleCount THEN
					simShuttleCount := 0;
					getShuttleStep := getShuttleADDWAIT;
				ELSE
					getShuttleStep := getShuttleLOADWAIT;
				END_IF;
			END_IF;

		getShuttleADDWAIT:
			// Füge ein Shuttle hinzu (nur Simulation!).
			FB_addShuttle.Position := simShuttleCount * 0.1;
			FB_addShuttle.Execute := TRUE;
			IF FB_addShuttle.Done THEN
				FB_addShuttle.Execute := FALSE;
				getShuttleStep := getShuttleADD;
			END_IF;

		getShuttleADD:
			// Zähle hoch und falls geforderte Anzahl erreicht, gehe weiter.
			simShuttleCount := simShuttleCount + 1;
			IF simShuttleCount = trakAsmb.cmd.simulation THEN
				getShuttleStep := getShuttleLOADWAIT;
			ELSE
				getShuttleStep := getShuttleADDWAIT;
			END_IF;

		getShuttleLOADWAIT:
			// Rufe GetShuttle FB auf und warte bis dieser fertig ist.
			FB_getShuttle.Enable := TRUE;
			FB_getShuttle.Next := TRUE;
			IF FB_getShuttle.Valid THEN
				getShuttleStep := getShuttleLOAD;
			END_IF;

		getShuttleLOAD:
			// Speichere Daten des geladenen Shuttles.
			trakAsmb.shuttles[FB_getShuttle.RemainingCount].axis := FB_getShuttle.Axis;
			trakAsmb.shuttles[FB_getShuttle.RemainingCount].id := FB_getShuttle.AdditionalInfo.ShuttleID;
			// Haben wir alle Shuttles gelesen?
			IF FB_getShuttle.RemainingCount <> 0 THEN
				// Nein, setze Next zurück, nächstes Laden eines Shuttles wird mit positiver Flanke im LOADWAIT ausgelöst.
				FB_getShuttle.Next := FALSE;
				getShuttleStep := getShuttleLOADWAIT;
			ELSE
				// Ja, wir sind fertig.
				getShuttleStep := getShuttleDONE;
				// speichere zudem die Anzahl gefundener Shuttles
				trakAsmb.shuttleCount := FB_getShuttle.TotalCount;
			END_IF;

		getShuttleDONE:
			// Alle Shuttles geladen, deaktiviere FB wir sind fertig.
			FB_getShuttle.Enable := FALSE;
			FB_getShuttle.Next := FALSE;
			// Lösche Befehl zum neuladen.
			trakAsmb.cmd.reload := FALSE;

	END_CASE;

	// Rufe alle FBs zyklisch auf, werden aber nur berechnet wenn "Enable" oder "Execute" aktiv.
	FB_status();
	FB_reset();
	FB_powerOff();
	FB_powerOn();
	FB_getShuttle();
	FB_addShuttle();

	// Enable der FBs deaktivieren wenn Busy Signal geht oder Fehler ansteht.
	IF EDGENEG(FB_reset.Busy) OR FB_reset.Error THEN
		FB_reset.Execute := FALSE;
		trakAsmb.cmd.reset := FALSE;
	END_IF;
	IF EDGENEG(FB_powerOff.Busy) OR FB_powerOff.Error THEN
		FB_powerOff.Execute := FALSE;
	END_IF;
	IF EDGENEG(FB_powerOn.Busy) OR FB_powerOn.Error THEN
		FB_powerOn.Execute := FALSE;
	END_IF;

END_PROGRAM

PROGRAM _EXIT
	(* Insert code here *)

END_PROGRAM
```

### Program Logical/TrakControl/trakConvoy (IEC)

#### Types.typ
```iecst
TYPE
	intFsmStep_t :
		(
		STEP_RESET,
		STEP_RESET_WAIT,
		STEP_RESET_MOVE,
		STEP_RESET_NEXT,
		STEP_IDLE,
		STEP_WAIT_MASTER,
		STEP_GET_MASTER,
		STEP_POS_MASTER,
		STEP_WAIT_SLAVE,
		STEP_GET_SLAVE,
		STEP_POS_SLAVE,
		STEP_PREPARED,
		STEP_CONVOY_CREATE,
		STEP_CONVOY_ADD,
		STEP_CONVOY_COUPLE,
		STEP_COUPLED,
		STEP_MOVE,
		STEP_MOVED,
		STEP_RELEASE_SLAVE,
		STEP_RELEASE_MASTER,
		STEP_RELEASED,
		STEP_RETURN_MASTER,
		STEP_RETURN_MASTER_WAIT,
		STEP_RETURN_SLAVE,
		STEP_RETURN_SLAVE_WAIT,
		STEP_RETURNED
		);
END_TYPE
```

#### Variables.var
```iecst
(*Schnittstelle nach aussen*)
VAR
	fsmStep : intFsmStep_t;
	distanceSet : LREAL;
	distanceActual : LREAL;
	masterAxis : McAxisType;
	slaveAxis : McAxisType;
	shuttleResetCounter : UINT;
END_VAR
(*Interne FBs*)
VAR
	FB_move : MC_BR_RoutedMoveAbs_AcpTrak;
	FB_createConvoy : MC_BR_ShCreateConvoy_AcpTrak;
	FB_add2Convoy : MC_BR_ShMoveInConvoy_AcpTrak;
	FB_deleteConvoy : MC_BR_ConDelete_AcpTrak;
	FB_moveVel : MC_BR_RoutedMoveVel_AcpTrak;
	FB_ppCommand : MC_BR_BarrierCommand_AcpTrak;
	FB_ppGet : MC_BR_BarrierGetShuttle_AcpTrak;
	New_Variable2 : USINT;
	New_Variable1 : USINT;
	New_Variable : USINT;
	FB_readSetMaster : MC_BR_ReadCyclicPosition;
	FB_readActMaster : MC_BR_ReadCyclicPosition;
	FB_readSetSlave : MC_BR_ReadCyclicPosition;
	FB_readActSlave : MC_BR_ReadCyclicPosition;
END_VAR
```

#### Main.st
```iecst
PROGRAM _INIT
	// Initialsiere alle FBs
	FB_move.Velocity      	:= 1.5;
	FB_move.Acceleration  	:= 10.0;
	FB_move.Deceleration  	:= 10.0;
	FB_move.Jerk          	:= 0.0;
	FB_move.BufferMode    	:= mcABORTING;
	FB_move.AdvancedParameters.StartDirection     := mcDIR_UNDEFINED;
	FB_move.AdvancedParameters.EndDirection       := mcDIR_POSITIVE;
	FB_move.AdvancedParameters.ShuttleOrientation := mcDIR_UNDEFINED;

	FB_moveVel.Velocity      	:= 1.5;
	FB_moveVel.Acceleration  	:= 10.0;
	FB_moveVel.Deceleration  	:= 10.0;
	FB_moveVel.Jerk          	:= 0.0;
	FB_moveVel.BufferMode    	:= mcABORTING;
	FB_moveVel.AdvancedParameters.StartDirection     := mcDIR_UNDEFINED;
	FB_moveVel.AdvancedParameters.EndDirection       := mcDIR_POSITIVE;
	FB_moveVel.AdvancedParameters.ShuttleOrientation := mcDIR_UNDEFINED;

	FB_createConvoy.Parameters.NegativeOffset := 0.2;
	FB_createConvoy.Parameters.PositiveOffset := 0.2;
	FB_createConvoy.Parameters.Separable := FALSE;
	FB_createConvoy.Parameters.Elastic := TRUE;
	//FB_createConvoy.Parameters.MasterVelocityAdjustment := TRUE;
	//FB_createConvoy.Parameters.TargetDistDeceleration := 0.0;

	FB_add2Convoy.Parameters.CouplingMode := mcACPTRAK_COUPL_DIST;
	FB_add2Convoy.Parameters.Elastic := TRUE;
	FB_add2Convoy.AdvancedParameters.Velocity := 4.0;
	FB_add2Convoy.AdvancedParameters.Acceleration := 20.0;
	FB_add2Convoy.AdvancedParameters.Deceleration := 20.0;
	FB_add2Convoy.AdvancedParameters.TargetDistance := -0.09; //0.126;

	FB_readActMaster.ValueSource := mcVALUE_ACTUAL;
	FB_readActSlave.ValueSource  := mcVALUE_ACTUAL;
	FB_readSetMaster.ValueSource := mcVALUE_SET;
	FB_readSetSlave.ValueSource  := mcVALUE_SET;

	FB_ppCommand.ProcessPoint := ADR(gPPDepot);
	FB_ppCommand.Command := mcACPTRAK_BARRIER_ADD_TICKETS;
	FB_ppCommand.AdvancedParameters.TicketCount := 2;
	//FB_ppCommand.AdvancedParameters.TicketCount := 1;

	FB_ppGet.ProcessPoint := ADR(gPPDepot);
	FB_ppGet.AdvancedParameters.SelectionMode := mcACPTRAK_BARR_GET_SH_CLOSEST;
	FB_ppGet.Next := FALSE;

	// alle FBs deaktivieren
	FB_move.Execute 		:= FALSE;
	FB_moveVel.Execute 		:= FALSE;
	FB_createConvoy.Execute := FALSE;
	FB_add2Convoy.Execute	:= FALSE;
	FB_deleteConvoy.Execute := FALSE;
	FB_readSetMaster.Enable := FALSE;
	FB_readActMaster.Enable := FALSE;
	FB_readSetSlave.Enable 	:= FALSE;
	FB_readActSlave.Enable 	:= FALSE;
	FB_ppCommand.Execute 	:= FALSE;

	// auslesen der Depot PP immer aktivieren
	FB_ppGet.Enable := TRUE;

	// Startzustand
	fsmStep := STEP_RESET;
	shuttleResetCounter := 0;

END_PROGRAM

PROGRAM _CYCLIC
	// Durchlaufe eine FSM um zwei Shuttles zu koppeln.
	CASE fsmStep OF
		STEP_RESET:
			// Depot Barriere Schliessen
			FB_ppCommand.Command := mcACPTRAK_BARRIER_CLOSE;
			FB_ppCommand.Execute := TRUE;
			// Weiter wenn Kommando ausgeführt wurde
			IF FB_ppCommand.Done THEN
				FB_ppCommand.Execute := FALSE;
				// Weiter
				fsmStep := STEP_RESET_WAIT;
			END_IF;

		STEP_RESET_WAIT:
			// Warte bis Assembly ready.
			IF trakAsmb.state.ready THEN
				shuttleResetCounter := 0;
				fsmStep := STEP_RESET_MOVE;
			END_IF;

		STEP_RESET_MOVE:
			// Alle Shuttles im Assembly ins Depot bewegen.
			FB_moveVel.Sector := ADR(gSecFull);
			FB_moveVel.Position := 6.0; // Position ist hinterhalb des PP gPPDepot (ist bei pos 5.6)
			FB_moveVel.Axis := ADR(trakAsmb.shuttles[shuttleResetCounter].axis);
			FB_moveVel.Execute := TRUE;
			// Direkt weiter sobald Fahrbefehl aktiv, wird im Hintergrund weitergeführt.
			IF EDGEPOS(FB_moveVel.Active) THEN
				FB_moveVel.Execute := FALSE;
				fsmStep := STEP_RESET_NEXT;
			END_IF;

		STEP_RESET_NEXT:
			// Nächstes Shuttle senden.
			shuttleResetCounter := shuttleResetCounter + 1;
			// Wenn Zähler die Anzahl Shuttles erreicht hat, sind wir fertig mit allen Shuttles.
			// Ansonsten zum nächsten Shuttle.
			IF shuttleResetCounter = trakAsmb.shuttleCount THEN
				fsmStep := STEP_IDLE;
			ELSE
				fsmStep := STEP_RESET_MOVE;
			END_IF;

		STEP_IDLE:
			// Warte auf Ready + Befehl.
			IF (trakConvoy.cmd.prepare AND trakAsmb.state.ready) THEN
				trakConvoy.cmd.prepare := FALSE;
				fsmStep := STEP_WAIT_MASTER;
			END_IF;

		STEP_WAIT_MASTER:
			// Warte bis ein Shuttle hinter der Barriere wartet
			IF (FB_ppGet.Valid AND FB_ppGet.TotalCount <> 0) THEN
				// Shuttle gefunden, speichere Achse
				masterAxis := FB_ppGet.Axis;
				// Aktiviere lesen des Master Position
				FB_readSetMaster.Axis := ADR(masterAxis);
				FB_readSetMaster.Enable := TRUE;
				FB_readActMaster.Axis := ADR(masterAxis);
				FB_readActMaster.Enable := TRUE;
				// Weiter
				fsmStep := STEP_GET_MASTER;
			END_IF;

		STEP_GET_MASTER:
			// Löse ein Shuttle aus dem Depot
			FB_ppCommand.AdvancedParameters.TicketCount := 1;
			FB_ppCommand.Command := mcACPTRAK_BARRIER_ADD_TICKETS;
			FB_ppCommand.Execute := TRUE;
			// Weiter wenn Kommando ausgeführt wurde
			IF FB_ppCommand.Done THEN
				FB_ppCommand.Execute := FALSE;
				fsmStep := STEP_POS_MASTER;
			END_IF;

		STEP_POS_MASTER:
			// Sende neue Sollposition
			FB_move.Sector := ADR(gSecFull);
			FB_move.Position := trakConvoy.startPos;
			FB_move.Axis := ADR(masterAxis);
			FB_move.Execute := TRUE;
			// Weiter wenn Bewegung abgeschlossen.
			IF FB_move.Done THEN
				FB_move.Execute := FALSE;
				fsmStep := STEP_WAIT_SLAVE;
			END_IF;

		STEP_WAIT_SLAVE:
			// Warte bis ein Shuttle hinter der Barriere wartet
			IF (FB_ppGet.Valid AND FB_ppGet.TotalCount <> 0) THEN
				// Shuttle gefunden, speichere Achse
				slaveAxis := FB_ppGet.Axis;
				// Aktiviere lesen des Slave Position
				FB_readSetSlave.Axis := ADR(slaveAxis);
				FB_readSetSlave.Enable := TRUE;
				FB_readActSlave.Axis := ADR(slaveAxis);
				FB_readActSlave.Enable := TRUE;
				// Weiter
				fsmStep := STEP_GET_SLAVE;
			END_IF;

		STEP_GET_SLAVE:
			// Löse ein Shuttle aus dem Depot
			FB_ppCommand.AdvancedParameters.TicketCount := 1;
			FB_ppCommand.Command := mcACPTRAK_BARRIER_ADD_TICKETS;
			FB_ppCommand.Execute := TRUE;
			// Weiter wenn Kommando ausgeführt wurde
			IF FB_ppCommand.Done THEN
				FB_ppCommand.Execute := FALSE;
				fsmStep := STEP_POS_SLAVE;
			END_IF;

		STEP_POS_SLAVE:
			// Sende neue Sollposition
			FB_move.Sector := ADR(gSecFull);
			FB_move.Position := trakConvoy.startPos - trakConvoy.coupleDistance - 0.01;
			FB_move.Axis := ADR(slaveAxis);
			FB_move.Execute := TRUE;
			// Weiter wenn Bewegung abgeschlossen.
			IF FB_move.Done THEN
				FB_move.Execute := FALSE;
				fsmStep := STEP_PREPARED;
			END_IF;

		STEP_PREPARED:
			// Warte auf Ready + Befehl.
			IF (trakConvoy.cmd.couple AND trakAsmb.state.ready) THEN
				trakConvoy.cmd.couple := FALSE;
				fsmStep := STEP_CONVOY_CREATE;
			END_IF;

		STEP_CONVOY_CREATE:
			// Erstelle Convoy
			FB_createConvoy.Axis := ADR(masterAxis);
			FB_createConvoy.Execute := TRUE;
			// Weiter wenn Convoy erstellt wurde
			IF FB_createConvoy.Done THEN
				FB_createConvoy.Execute := FALSE;
				fsmStep := STEP_CONVOY_ADD;
			END_IF;

		STEP_CONVOY_ADD:
			// Slave dem Convoy hinzufügen
			FB_add2Convoy.Parameters.ReferenceShuttle := ADR(masterAxis); // master
			FB_add2Convoy.Axis := ADR(slaveAxis); // slave
			FB_add2Convoy.Execute := TRUE;
			// Weiter wenn an Convoy angeschlossen
			IF FB_add2Convoy.Done THEN
				FB_add2Convoy.Execute := FALSE;
				fsmStep := STEP_CONVOY_COUPLE;
			END_IF;

		STEP_CONVOY_COUPLE:
			// Pseudo koppeln. Durch Convoy sind Shuttles bereits gekoppelt aber Convoy wurde erst gerade erstellt.
			// Mit einem Move Befehl den Master auf der aktuellen Position (+kleiner Offset) neu positionieren, dies
			// sollte gesamtes Convoy neu ausrichten bez. die eingestellten Abstände einstellen.
			// Sende neue Sollposition
			FB_move.Sector := ADR(gSecFull);
			FB_move.Position := trakConvoy.startPos + 0.01;
			FB_move.Axis := ADR(masterAxis);
			FB_move.Execute := TRUE;
			// Weiter wenn Bewegung abgeschlossen.
			IF FB_move.Done THEN
				FB_move.Execute := FALSE;
				fsmStep := STEP_COUPLED;
			END_IF;

		STEP_COUPLED:
			// Warte auf Ready + Befehl.
			IF (trakConvoy.cmd.move AND trakAsmb.state.ready) THEN
				trakConvoy.cmd.move := FALSE;
				fsmStep := STEP_MOVE;
			END_IF;

		STEP_MOVE:
			FB_move.Sector := ADR(gSecFull);
			FB_move.Position := trakConvoy.targetPos;
			FB_move.Axis := ADR(masterAxis);
			FB_move.Execute := TRUE;
			// Weiter wenn Bewegung abgeschlossen.
			IF FB_move.Done THEN
				FB_move.Execute := FALSE;
				fsmStep := STEP_MOVED;
			END_IF;

		STEP_MOVED:
			// Warte auf Ready + Befehl.
			IF (trakConvoy.cmd.release AND trakAsmb.state.ready) THEN
				trakConvoy.cmd.release := FALSE;
				fsmStep := STEP_RELEASE_SLAVE;
			END_IF;

		STEP_RELEASE_SLAVE:
			// Entferne Slave aus dem Convoy mittels Bewegungsbefehl.
			FB_move.Sector := ADR(gSecFull);
			FB_move.Position := trakConvoy.targetPos - trakConvoy.coupleDistance - 0.01;
			FB_move.AdvancedParameters.EndDirection := mcDIR_NEGATIVE; // fahre rückwärts!
			FB_move.Axis := ADR(slaveAxis);
			FB_move.Execute := TRUE;
			// Weiter wenn Bewegung abgeschlossen.
			IF FB_move.Done THEN
				FB_move.Execute := FALSE;
				FB_move.AdvancedParameters.EndDirection := mcDIR_POSITIVE;
				fsmStep := STEP_RELEASE_MASTER;
			END_IF;

		STEP_RELEASE_MASTER:
			// Löse Convoy auf.
			FB_deleteConvoy.ConvoyMaster := ADR(masterAxis);
			FB_deleteConvoy.Execute := TRUE;
			// Weiter wenn Convoy aufgelöst.
			IF FB_deleteConvoy.Done THEN
				FB_deleteConvoy.Execute := FALSE;
				fsmStep := STEP_RELEASED;
			END_IF;

		STEP_RELEASED:
			// Warte auf Ready + Befehl.
			IF (trakConvoy.cmd.return AND trakAsmb.state.ready) THEN
				trakConvoy.cmd.return := FALSE;
				fsmStep := STEP_RETURN_MASTER;
			END_IF;

		STEP_RETURN_MASTER:
			FB_moveVel.Sector := ADR(gSecFull);
			FB_moveVel.Position := 6.0; // Position ist hinterhalb des PP gPPDepot (ist bei pos 5.6)
			FB_moveVel.Axis := ADR(masterAxis);
			FB_moveVel.Execute := TRUE;
			// Direkt weiter.
			fsmStep := STEP_RETURN_MASTER_WAIT;

		STEP_RETURN_MASTER_WAIT:
			// Direkt weiter sobald Fahrbefehl aktiv, wird im Hintergrund weitergeführt.
			IF FB_moveVel.Active THEN
				FB_moveVel.Execute := FALSE;
				fsmStep := STEP_RETURN_SLAVE;
			END_IF;

		STEP_RETURN_SLAVE:
			FB_moveVel.Sector := ADR(gSecFull);
			FB_moveVel.Position := 6.0; // Position ist hinterhalb des PP gPPDepot (ist bei pos 5.6)
			FB_moveVel.Axis := ADR(slaveAxis);
			FB_moveVel.Execute := TRUE;
			// Direkt weiter.
			fsmStep := STEP_RETURN_SLAVE_WAIT;

		STEP_RETURN_SLAVE_WAIT:
			// Direkt weiter sobald Fahrbefehl aktiv, wird im Hintergrund weitergeführt.
			IF FB_moveVel.Active THEN
				FB_moveVel.Execute := FALSE;
				fsmStep := STEP_RETURNED;
			END_IF;

		STEP_RETURNED:
			// Dummy step, gehe zurück in Start. Shuttles sind ggf. noch unterwegs ins Depot.
			fsmStep := STEP_IDLE;

	END_CASE;

	// Status zurückmelden
	trakConvoy.state.prepared := (fsmStep = STEP_PREPARED);
	trakConvoy.state.coupled  := (fsmStep = STEP_COUPLED);
	trakConvoy.state.moved    := (fsmStep = STEP_MOVED);
	trakConvoy.state.released := (fsmStep = STEP_RELEASED);
	trakConvoy.state.returned := (fsmStep = STEP_RETURNED OR fsmStep = STEP_IDLE);

	// Alle Bewegungs-FBs deaktivieren wenn Assembly nicht ready ist.
	IF NOT trakAsmb.state.ready THEN
		FB_move.Execute := FALSE;
		FB_moveVel.Execute := FALSE;
	END_IF;

	// Bei Reset Kommando alle Bewegungs-FBs deaktivieren und Zustand wechseln.
	IF trakConvoy.cmd.reset THEN
		FB_move.Execute := FALSE;
		FB_moveVel.Execute := FALSE;
		trakConvoy.cmd.reset := FALSE;
		fsmStep := STEP_RESET;
	END_IF;

	// Rufe alle FBs zyklisch auf, werden aber nur berechnet wenn "Enable" oder "Execute" aktiv.
	FB_move();
	FB_moveVel();
	FB_createConvoy();
	FB_add2Convoy();
	FB_deleteConvoy();
	FB_readSetMaster();
	FB_readActMaster();
	FB_readSetSlave();
	FB_readActSlave();
	FB_ppCommand();
	FB_ppGet();

	distanceActual := FB_readActMaster.CyclicPosition - FB_readActSlave.CyclicPosition;
	distanceSet := FB_readSetMaster.CyclicPosition - FB_readSetSlave.CyclicPosition;

	// Enable der FBs deaktivieren wenn Busy Signal geht oder Fehler ansteht.
	//IF EDGENEG(FB_move.Busy) OR FB_move.Error THEN
	//	FB_move.Execute := FALSE;
	//END_IF;
	//IF EDGENEG(FB_couple.Busy) OR FB_couple.Error THEN
	//	FB_couple.Execute := FALSE;
	//END_IF;

END_PROGRAM

PROGRAM _EXIT
	(* Insert code here *)

END_PROGRAM
```

### Program Logical/TrakControl/trakCouple (IEC)

#### Types.typ
```iecst
TYPE
	trakMoveCmd_t : 	STRUCT
		trace : BOOL;
		test : BOOL;
	END_STRUCT;
	trakMove_t : 	STRUCT
		cmd : trakMoveCmd_t;
	END_STRUCT;
	intCoupleStep_t :
		(
		coupleStepWAIT,
		coupleStepSENDPOS1,
		coupleStepSENDPOS2,
		coupleStepSETOBJ1,
		coupleStepSETOBJ2,
		coupleStepCOUPLE,
		coupleStepDONE
	);
END_TYPE
```

#### Variables.var
```iecst
(*Schnittstelle nach aussen*)
VAR
	dummyFirst : UINT;
	dummySecond : UINT;
	trakMove : trakMove_t;
	coupleStep : intCoupleStep_t;
	distanceSet : LREAL;
	distanceActual : LREAL;
END_VAR
(*Interne FBs*)
VAR
	FB_move : MC_BR_RoutedMoveAbs_AcpTrak;
	FB_couple : MC_BR_ShCouplingObjCmd_AcpTrak;
	FB_gearin : MC_GearIn;
	FB_moveVel : MC_BR_RoutedMoveVel_AcpTrak;
	FB_moveCyc : MC_BR_ElasticMoveCycPos_AcpTrak;
	FB_read1 : MC_BR_ReadCyclicPosition;
	FB_read2 : MC_BR_ReadCyclicPosition;
	FB_read3 : MC_BR_ReadCyclicPosition;
	FB_read4 : MC_BR_ReadCyclicPosition;
END_VAR
```

#### Main.st
```iecst
PROGRAM _INIT
	// Initialsiere alle FBs
	FB_move.Velocity      	:= 0.8;
	FB_move.Acceleration  	:= 10.0;
	FB_move.Deceleration  	:= 10.0;
	FB_move.Jerk          	:= 0.0;
	FB_move.BufferMode    	:= mcABORTING;
	FB_move.AdvancedParameters.StartDirection     := mcDIR_UNDEFINED;
	FB_move.AdvancedParameters.EndDirection       := mcDIR_POSITIVE;
	FB_move.AdvancedParameters.ShuttleOrientation := mcDIR_UNDEFINED;

	FB_couple.Command := mcACPTRAK_COUPLE_OBJ_SET;

	FB_gearin.RatioNumerator 	:= 1; // synchrone 1:1 Bewegung
	FB_gearin.RatioDenominator 	:= 1;
	FB_gearin.Acceleration 		:= 0.0; // nutze Maximalerte des Slaves
	FB_gearin.Deceleration 		:= 0.0;
	FB_gearin.Jerk 				:= 0.0;
	FB_gearin.BufferMode 		:= mcABORTING;
	FB_gearin.MasterValueSource := mcVALUE_ACTUAL;

	FB_moveVel.Velocity      	:= 0.8;
	FB_moveVel.RouteVelocity	:= 0.8;
	FB_moveVel.Acceleration  	:= 2.0;
	FB_moveVel.Deceleration  	:= 2.0;
	FB_moveVel.Jerk          	:= 0.0;
	FB_moveVel.BufferMode    	:= mcABORTING;
	FB_moveVel.AdvancedParameters.StartDirection     := mcDIR_UNDEFINED;
	FB_moveVel.AdvancedParameters.EndDirection       := mcDIR_POSITIVE;
	FB_moveVel.AdvancedParameters.ShuttleOrientation := mcDIR_UNDEFINED;

	FB_moveCyc.InterpolationMode 	:= mcIPLM_DEFAULT;
	FB_moveCyc.CyclicPosition 		:= 1.0;
	FB_moveCyc.AdvancedParameters.Velocity 		:= 0.8;
	FB_moveCyc.AdvancedParameters.Acceleration 	:= 2.0;
	FB_moveCyc.AdvancedParameters.Deceleration 	:= 2.0;
	FB_moveCyc.AdvancedParameters.Jerk			:= 0.0;

	FB_read1.ValueSource := mcVALUE_ACTUAL;
	FB_read2.ValueSource := mcVALUE_ACTUAL;
	FB_read3.ValueSource := mcVALUE_SET;
	FB_read4.ValueSource := mcVALUE_SET;

	// alle FBs deaktivieren
	FB_move.Execute 	:= FALSE;
	FB_couple.Execute 	:= FALSE;
	FB_gearin.Execute 	:= FALSE;
	FB_moveVel.Execute 	:= FALSE;
	FB_moveCyc.Enable 	:= FALSE;
	FB_read1.Enable 	:= FALSE;
	FB_read2.Enable 	:= FALSE;
	FB_read3.Enable 	:= FALSE;
	FB_read4.Enable 	:= FALSE;

	dummyFirst := 1;
	dummySecond := 0;

END_PROGRAM

PROGRAM _CYCLIC
	// Durchlaufe eine FSM um zwei Shuttles zu verbinden.
	CASE coupleStep OF
		coupleStepWAIT:
			// Warte auf Ready + Befehl.
			IF (trakMove.cmd.test AND trakAsmb.state.ready) THEN
				coupleStep := coupleStepSENDPOS1;
				trakMove.cmd.test := FALSE;
			END_IF;

		coupleStepSENDPOS1:
			// Starte Bewegung des ersten Shuttles.
			FB_move.Sector := ADR(gSecFull);
			FB_move.Position := 0.426;
			FB_move.Axis := ADR(trakAsmb.shuttles[dummyFirst].axis);
			FB_move.Execute := TRUE;
			// Weiter wenn Bewegung abgeschlossen.
			IF FB_move.Done THEN
				FB_move.Execute := FALSE;
				coupleStep := coupleStepSENDPOS2;
			END_IF;

		coupleStepSENDPOS2:
			// Starte Bewegung des zweiten Shuttles.
			FB_move.Sector := ADR(gSecFull);
			FB_move.Position := 0.3;
			FB_move.Axis := ADR(trakAsmb.shuttles[dummySecond].axis);
			FB_move.Execute := TRUE;
			// Weiter wenn Bewegung abgeschlossen.
			IF FB_move.Done THEN
				FB_move.Execute := FALSE;
				coupleStep := coupleStepSETOBJ1;
			END_IF;

		coupleStepSETOBJ1:
			// Manueller Schritt, setze coupleStep per PV Watch auf coupleStepSETOBJ2
			// DEBUG: Skip
			//coupleStep := coupleStepCOUPLE;

		coupleStepSETOBJ2:
			// TEST
			FB_read1.Axis := ADR(trakAsmb.shuttles[dummyFirst].axis);
			FB_read2.Axis := ADR(trakAsmb.shuttles[dummySecond].axis);
			FB_read1.Enable := TRUE;
			FB_read2.Enable := TRUE;
			FB_read3.Axis := ADR(trakAsmb.shuttles[dummyFirst].axis);
			FB_read4.Axis := ADR(trakAsmb.shuttles[dummySecond].axis);
			FB_read3.Enable := TRUE;
			FB_read4.Enable := TRUE;
			// Kopplungsobjekt an zweites Shuttle h?ngen
			FB_couple.Axis := ADR(trakAsmb.shuttles[dummySecond].axis);
			FB_couple.CouplingObjectName := 'couplingLoad';
			FB_couple.Execute := TRUE;
			// Weiter wenn an Objekt angeschlossen.
			IF FB_couple.Done THEN
				FB_couple.Execute := FALSE;
				coupleStep := coupleStepCOUPLE;
			END_IF;

		coupleStepCOUPLE:
			// Achsen synchronisieren bez. tats?chlich Koppeln.
			FB_gearin.Master := ADR(trakAsmb.shuttles[dummyFirst].axis);
			FB_gearin.Slave := ADR(trakAsmb.shuttles[dummySecond].axis);
			FB_gearin.Execute := TRUE;
			// Wenn Kopplung aktiv ist, dann sind wir fertig.
			IF FB_gearin.Active THEN
				coupleStep := coupleStepDONE;
			END_IF;

		coupleStepDONE:
			// Master Shuttle bewegen.
			FB_moveCyc.Axis := ADR(trakAsmb.shuttles[dummyFirst].axis);
			FB_moveCyc.Enable := TRUE;
		// Weiter wenn Bewegung abgeschlossen.
		//IF FB_moveCyc.Done THEN
		//	FB_moveAdd.Execute := FALSE;
		//	coupleStep := coupleStepWAIT;
		//END_IF;

	END_CASE;

	// Rufe alle FBs zyklisch auf, werden aber nur berechnet wenn "Enable" oder "Execute" aktiv.
	FB_move();
	FB_couple();
	FB_gearin();
	FB_moveVel();
	FB_moveCyc();
	FB_read1();
	FB_read2();
	FB_read3();
	FB_read4();

	distanceActual := FB_read1.CyclicPosition - FB_read2.CyclicPosition;
	distanceSet := FB_read3.CyclicPosition - FB_read4.CyclicPosition;

	// Enable der FBs deaktivieren wenn Busy Signal geht oder Fehler ansteht.
	//IF EDGENEG(FB_move.Busy) OR FB_move.Error THEN
	//	FB_move.Execute := FALSE;
	//END_IF;
	//IF EDGENEG(FB_couple.Busy) OR FB_couple.Error THEN
	//	FB_couple.Execute := FALSE;
	//END_IF;

	// Sobald Fehler in GearIn (keine Sanchronisation mehr) auftritt, dann stoppe komplettes Assembly
	IF FB_gearin.Error THEN
		trakAsmb.cmd.power := FALSE;
	END_IF;

END_PROGRAM

PROGRAM _EXIT
	(* Insert code here *)

END_PROGRAM
```

### Program Logical/TrakControl/trakSingle (IEC)

#### Types.typ
```iecst
TYPE
	intSingleStep_t :
		(
		singleStepIDLE,
		singleStepMOVE_ABB,
		singleStepWAIT_ABB,
		singleStepMOVE_DELTA,
		singleStepWAIT_DELTA
		);
END_TYPE
```

#### Variables.var
```iecst
(*Schnittstelle nach aussen*)
VAR
	positionSet : LREAL;
	positionActual : LREAL;
END_VAR
(*Interne FBs*)
VAR
	FB_move : MC_BR_RoutedMoveAbs_AcpTrak;
	FB_readSet : MC_BR_ReadCyclicPosition;
	FB_readActual : MC_BR_ReadCyclicPosition;
END_VAR
(*Interne Variablen*)
VAR
	posABB : LREAL := 0.272; (*Position auf Sektor gSecMajor*)
	posDelta : LREAL := 1.2; (*Position auf Sektor gSecMajor*)
	intSingleStep : intSingleStep_t;
END_VAR
```

#### Main.st
```iecst
PROGRAM _INIT
	// Initialsiere alle FBs
	FB_move.Velocity      	:= 0.8;
	FB_move.Acceleration  	:= 10.0;
	FB_move.Deceleration  	:= 10.0;
	FB_move.Jerk          	:= 0.0;
	FB_move.BufferMode    	:= mcABORTING;
	FB_move.AdvancedParameters.StartDirection     := mcDIR_UNDEFINED;
	FB_move.AdvancedParameters.EndDirection       := mcDIR_POSITIVE;
	FB_move.AdvancedParameters.ShuttleOrientation := mcDIR_UNDEFINED;

	FB_readSet.ValueSource 		:= mcVALUE_SET;
	FB_readActual.ValueSource	:= mcVALUE_ACTUAL;

	// alle FBs deaktivieren
	FB_move.Execute 	:= FALSE;
	FB_readSet.Enable 	:= FALSE;
	FB_readActual.Enable:= FALSE;

	// Initiale Zustände setzen
	trakSingle.cmd.goABB := FALSE;
	trakSingle.cmd.goDelta := FALSE;
	trakSingle.cmd.read := FALSE;
	trakSingle.state.atABB := FALSE;
	trakSingle.state.atDelta := FALSE;

END_PROGRAM

PROGRAM _CYCLIC
	// Lese die Position aus.
	FB_readSet.Enable    := trakSingle.cmd.read;
	FB_readActual.Enable := trakSingle.cmd.read;
	FB_readSet.Axis 	 := ADR(trakAsmb.shuttles[0].axis);
	FB_readActual.Axis 	 := ADR(trakAsmb.shuttles[0].axis);

	// Bewege Shuttle zu ABB oder Delta Position per FSM
	CASE intSingleStep OF
		singleStepIDLE:
			// Warte auf Fahrbefehl
			IF trakSingle.cmd.goABB THEN
				intSingleStep := singleStepMOVE_ABB;
			ELSIF trakSingle.cmd.goDelta THEN
				intSingleStep := singleStepMOVE_DELTA;
			END_IF;

		singleStepMOVE_ABB:
			// Starte Bewegung zur ABB Position
			FB_move.Axis := ADR(trakAsmb.shuttles[0].axis);
			FB_move.Sector := ADR(gSecMajor);
			FB_move.Position := posABB;
			FB_move.Execute := TRUE;
			trakSingle.state.atDelta := FALSE;
			intSingleStep := singleStepWAIT_ABB;

		singleStepWAIT_ABB:
			// Warte bis Position erreicht
			IF FB_move.Done THEN
				FB_move.Execute := FALSE;
				trakSingle.state.atABB := TRUE;
				intSingleStep := singleStepIDLE;
			END_IF;

		singleStepMOVE_DELTA:
			// Starte Bewegung zur Delta Position
			FB_move.Axis := ADR(trakAsmb.shuttles[0].axis);
			FB_move.Sector := ADR(gSecMajor);
			FB_move.Position := posDelta;
			FB_move.Execute := TRUE;
			trakSingle.state.atABB := FALSE;
			intSingleStep := singleStepWAIT_DELTA;

		singleStepWAIT_DELTA:
			// Warte bis Position erreicht
			IF FB_move.Done THEN
				FB_move.Execute := FALSE;
				trakSingle.state.atDelta := TRUE;
				intSingleStep := singleStepIDLE;
			END_IF;

	END_CASE;

	// Rufe alle FBs zyklisch auf, werden aber nur berechnet wenn "Enable" oder "Execute" aktiv.
	FB_move();
	FB_readSet();
	FB_readActual();

	positionSet := FB_readSet.CyclicPosition;
	positionActual := FB_readActual.CyclicPosition;

	trakSingle.state.moving := FB_move.Busy;

	// Bewegungsbefehle zurücksetzen wenn Bewegung aktiv
	IF FB_move.Busy THEN
		trakSingle.cmd.goABB := FALSE;
		trakSingle.cmd.goDelta := FALSE;
	END_IF;

END_PROGRAM

PROGRAM _EXIT
	(* Insert code here *)

END_PROGRAM
```

### Program Logical/TrakControl/trakFSM

#### Types.typ
```iecst
TYPE
	intGetShuttleStep_t :
		( (*Interner Schrittzustand des Shuttle-Get Befehls*)
		getShuttleRESET, (*Reset des trakShuttle Array Struktur*)
		getShuttleWAIT, (*Warte auf Ready des Assembly*)
		getShuttleADDWAIT, (*Simulation: Füge Shuttles hinzu*)
		getShuttleADD,
		getShuttleLOADWAIT, (*Triggere das Laden eines Shuttles*)
		getShuttleLOAD, (*Shuttle geladen, speichere seine Referenz*)
		getShuttleDONE (*Alle Shuttle Referenzen gespeichert, fertig.*)
		);
END_TYPE
```

#### Main.st
```iecst
PROGRAM _INIT
	// Initialsiere alle FBs
	FB_status.Assembly := ADR(gAssemblyFigure8);
	FB_reset.Assembly := ADR(gAssemblyFigure8);
	FB_powerOff.Assembly := ADR(gAssemblyFigure8);
	FB_powerOn.Assembly := ADR(gAssemblyFigure8);
	FB_getShuttle.Assembly := ADR(gAssemblyFigure8);
	FB_addShuttle.Sector := ADR(gSecMinor);
	FB_addShuttle.Sector := ADR(gDummyAxis);
	FB_addShuttle.Sector := ADR(gSecMajor);
	FB_addShuttle.Sector := ADR(gSecFull);

	// alle FBs ausser status deaktivieren
	FB_reset.Execute := FALSE;
	FB_powerOff.Execute := FALSE;
	FB_powerOn.Execute := FALSE;
	FB_getShuttle.Enable := FALSE;

	// Status FB aktivieren
	FB_status.Enable := TRUE;

	// Shuttle-Get FSM auf Reset
	getShuttleStep := getShuttleRESET;
	simShuttleCount := 0;

END_PROGRAM

PROGRAM _CYCLIC
	// Was ist der Zustand des Assembly?
	trakAsmb.state.errorStop := FB_status.AssemblyErrorStop;
	trakAsmb.state.disabled := FB_status.AssemblyDisabled;
	trakAsmb.state.homing := FB_status.AssemblyHoming;
	trakAsmb.state.stopping := FB_status.AssemblyStopping;
	// Wir sind die Shuttles am laden wenn Assembly bereit, aber Shuttle-Get FSM noch nicht.
	trakAsmb.state.loading := FB_status.AssemblyReady AND (getShuttleStep <> getShuttleDONE) AND getShuttleStep > getShuttleWAIT;
	// Wir sind komplett Bereit wenn Assembly und Shuttle-Get FSM bereit.
	trakAsmb.state.ready := FB_status.AssemblyReady AND getShuttleStep = getShuttleDONE;

	// Einschaltbefehl zurücksetzen wenn Zustand Ready verlassen wird.
	IF EDGENEG(FB_status.AssemblyReady) THEN
		trakAsmb.cmd.power := FALSE;
	END_IF;

	// Sind wir im Error oder wollen wir manuell Zurücksetzen? => Assembly zurücksetzen
	IF trakAsmb.state.errorStop OR trakAsmb.cmd.reset THEN
		FB_reset.Execute := TRUE;
		getShuttleStep := getShuttleRESET;
		trakAsmb.cmd.power := FALSE;
	END_IF;

	// Nach Reset kommen wir in Disabled, mit Einschaltbefehl ein PowerOn durchführen.
	IF trakAsmb.state.disabled AND trakAsmb.cmd.power THEN
		FB_powerOn.Execute := TRUE;
	END_IF;

	// Sind wir in Homing/Loading/Ready aber ohne Einschaltbefehl? => Stoppe Assembly
	IF (trakAsmb.state.homing OR trakAsmb.state.loading OR trakAsmb.state.ready) AND NOT trakAsmb.cmd.power THEN
		FB_powerOff.Execute := TRUE;
	END_IF;

	// Befehl zum Neuladen der Shuttles erhalten? => Get-Shuttle FSM zurücksetzen.
	IF (trakAsmb.cmd.reload AND getShuttleStep = getShuttleDONE) THEN
		getShuttleStep := getShuttleRESET;
		trakAsmb.cmd.reload := FALSE;
	END_IF;

	// Durchlaufe eine FSM um die Shuttlereferenzen per getShuttle FB zu erhalten.
	CASE getShuttleStep OF
		getShuttleRESET:
			// lösche die komplette Referenzstruktur
			brsmemset(ADR(trakAsmb.shuttles), 0, SIZEOF(trakAsmb.shuttles));
			trakAsmb.shuttleCount := 0;
			// warte auf nächsten Wechsel in Ready
			getShuttleStep := getShuttleWAIT;

		getShuttleWAIT:
			// Warte bis Assembly in Zustand Ready übergeht.
			IF FB_status.AssemblyReady THEN
				//getShuttleStep := getShuttleLOADWAIT;
				getShuttleStep := getShuttleADDWAIT;
			END_IF;

		getShuttleADDWAIT:
			trakAsmb.shuttleCount := 2;
			// Füge ein Shuttle hinzu (nur Simulation!), trakAsmb.shuttleCount dient als Anzahl der Shuttles.
			FB_addShuttle.Position := simShuttleCount * 0.1;
			FB_addShuttle.Execute := TRUE;
			IF FB_addShuttle.Done THEN
				FB_addShuttle.Execute := FALSE;
				getShuttleStep := getShuttleADD;
			END_IF;

		getShuttleADD:
			// Zähle hoch und falls geforderte Anzahl erreicht, gehe weiter.
			simShuttleCount := simShuttleCount + 1;
			IF simShuttleCount = trakAsmb.shuttleCount THEN
				getShuttleStep := getShuttleLOADWAIT;
			ELSE
				getShuttleStep := getShuttleADDWAIT;
			END_IF;

		getShuttleLOADWAIT:
			// Rufe GetShuttle FB auf und warte bis dieser fertig ist.
			FB_getShuttle.Enable := TRUE;
			FB_getShuttle.Next := TRUE;
			IF FB_getShuttle.Valid THEN
				getShuttleStep := getShuttleLOAD;
			END_IF;

		getShuttleLOAD:
			// Speichere Daten des geladenen Shuttles.
			trakAsmb.shuttles[FB_getShuttle.RemainingCount].axis := FB_getShuttle.Axis;
			trakAsmb.shuttles[FB_getShuttle.RemainingCount].id := FB_getShuttle.AdditionalInfo.ShuttleID;
			// Haben wir alle Shuttles gelesen?
			IF FB_getShuttle.RemainingCount <> 0 THEN
				// Nein, setze Next zurück, nächstes Laden eines Shuttles wird mit positiver Flanke im LOADWAIT ausgelöst.
				FB_getShuttle.Next := FALSE;
				getShuttleStep := getShuttleLOADWAIT;
			ELSE
				// Ja, wir sind fertig.
				getShuttleStep := getShuttleDONE;
				// speichere zudem die Anzahl gefundener Shuttles
				trakAsmb.shuttleCount := FB_getShuttle.TotalCount;
			END_IF;

		getShuttleDONE:
			// Alle Shuttles geladen, deaktiviere FB wir sind fertig.
			FB_getShuttle.Enable := FALSE;
			FB_getShuttle.Next := FALSE;
			// Lösche Befehl zum neuladen.
			trakAsmb.cmd.reload := FALSE;

	END_CASE;

	// Rufe alle FBs zyklisch auf, werden aber nur berechnet wenn "Enable" oder "Execute" aktiv.
	FB_status();
	FB_reset();
	FB_powerOff();
	FB_powerOn();
	FB_getShuttle();
	FB_addShuttle();

	// Enable der FBs deaktivieren wenn Busy Signal geht oder Fehler ansteht.
	IF EDGENEG(FB_reset.Busy) OR FB_reset.Error THEN
		FB_reset.Execute := FALSE;
		trakAsmb.cmd.reset := FALSE;
	END_IF;
	IF EDGENEG(FB_powerOff.Busy) OR FB_powerOff.Error THEN
		FB_powerOff.Execute := FALSE;
	END_IF;
	IF EDGENEG(FB_powerOn.Busy) OR FB_powerOn.Error THEN
		FB_powerOn.Execute := FALSE;
	END_IF;

END_PROGRAM

PROGRAM _EXIT
	(* Insert code here *)

END_PROGRAM
```

### Program Logical/TrakControl/trakMove

#### Types.typ
```iecst
TYPE
	trakMoveCmd_t : 	STRUCT
		trace : BOOL;
		test : BOOL;
	END_STRUCT;
	trakMove_t : 	STRUCT
		cmd : trakMoveCmd_t;
	END_STRUCT;
	intCoupleStep_t :
		(
		coupleStepWAIT,
		coupleStepSENDPOS1,
		coupleStepSENDPOS2,
		coupleStepSETOBJ1,
		coupleStepSETOBJ2,
		coupleStepCOUPLE,
		coupleStepDONE
		);
END_TYPE
```

#### Variables.var
```iecst
(*Schnittstelle nach aussen*)
VAR
	dummyFirst : UINT;
	dummySecond : UINT;
	trakMove : trakMove_t;
	coupleStep : intCoupleStep_t;
	distance : LREAL;
END_VAR
(*Interne FBs*)
VAR
	FB_move : MC_BR_RoutedMoveAbs_AcpTrak;
	FB_couple : MC_BR_ShCouplingObjCmd_AcpTrak;
	FB_gearin : MC_GearIn;
	FB_moveVel : MC_BR_RoutedMoveVel_AcpTrak;
	FB_moveCyc : MC_BR_ElasticMoveCycPos_AcpTrak;
	FB_createConvoy : MC_BR_ShCreateConvoy_AcpTrak;
	FB_add2Convoy : MC_BR_ShMoveInConvoy_AcpTrak;
	New_Variable1 : USINT;
	New_Variable : USINT;
	FB_read1 : MC_BR_ReadCyclicPosition;
	FB_read2 : MC_BR_ReadCyclicPosition;
END_VAR
```

#### Main.st
```iecst
PROGRAM _INIT
	// Initialsiere alle FBs
	FB_move.Velocity      	:= 0.8;
	FB_move.Acceleration  	:= 10.0;
	FB_move.Deceleration  	:= 10.0;
	FB_move.Jerk          	:= 0.0;
	FB_move.BufferMode    	:= mcABORTING;
	FB_move.AdvancedParameters.StartDirection     := mcDIR_UNDEFINED;
	FB_move.AdvancedParameters.EndDirection       := mcDIR_POSITIVE;
	FB_move.AdvancedParameters.ShuttleOrientation := mcDIR_UNDEFINED;

	//FB_couple.Command := mcACPTRAK_COUPLE_OBJ_SET;

	//FB_gearin.Master 			:= ADR(gDummyAxis);
	//FB_gearin.RatioNumerator 	:= 1; // synchrone 1:1 Bewegung
	//FB_gearin.RatioDenominator 	:= 1;
	//FB_gearin.Acceleration 		:= 0.0; // nutze Maximalerte des Slaves
	//FB_gearin.Deceleration 		:= 0.0;
	//FB_gearin.Jerk 				:= 0.0;
	//FB_gearin.BufferMode 		:= mcABORTING;
	//FB_gearin.MasterValueSource := mcVALUE_ACTUAL;

	FB_moveVel.Velocity      	:= 0.8;
	FB_moveVel.RouteVelocity	:= 0.8;
	FB_moveVel.Acceleration  	:= 2.0;
	FB_moveVel.Deceleration  	:= 2.0;
	FB_moveVel.Jerk          	:= 0.0;
	FB_moveVel.BufferMode    	:= mcABORTING;
	FB_moveVel.AdvancedParameters.StartDirection     := mcDIR_UNDEFINED;
	FB_moveVel.AdvancedParameters.EndDirection       := mcDIR_POSITIVE;
	FB_moveVel.AdvancedParameters.ShuttleOrientation := mcDIR_UNDEFINED;

	FB_moveCyc.InterpolationMode 	:= mcIPLM_DEFAULT;
	FB_moveCyc.CyclicPosition 		:= 1.0;
	FB_moveCyc.AdvancedParameters.Velocity 		:= 0.8;
	FB_moveCyc.AdvancedParameters.Acceleration 	:= 2.0;
	FB_moveCyc.AdvancedParameters.Deceleration 	:= 2.0;
	FB_moveCyc.AdvancedParameters.Jerk			:= 0.0;

	FB_createConvoy.Parameters.NegativeOffset := 0.0;
	FB_createConvoy.Parameters.PositiveOffset := 0.2;
	FB_createConvoy.Parameters.Separable := FALSE;
	FB_createConvoy.Parameters.Elastic := TRUE;

	FB_add2Convoy.Parameters.CouplingMode := mcACPTRAK_COUPL_DIST;
	FB_add2Convoy.Parameters.Elastic := TRUE;
	FB_add2Convoy.AdvancedParameters.Velocity := 4.0;
	FB_add2Convoy.AdvancedParameters.Acceleration := 20.0;
	FB_add2Convoy.AdvancedParameters.Deceleration := 20.0;
	FB_add2Convoy.AdvancedParameters.TargetDistance := 0.126;

	FB_read1.ValueSource := mcVALUE_ACTUAL;
	FB_read2.ValueSource := mcVALUE_ACTUAL;

	// alle FBs deaktivieren
	FB_move.Execute 	:= FALSE;
	FB_couple.Execute 	:= FALSE;
	FB_gearin.Execute 	:= FALSE;
	FB_moveVel.Execute 	:= FALSE;
	FB_moveCyc.Enable 	:= FALSE;
	FB_createConvoy.Execute := FALSE;
	FB_read1.Enable 	:= FALSE;
	FB_read2.Enable 	:= FALSE;

	dummyFirst := 1;
	dummySecond := 0;

END_PROGRAM

PROGRAM _CYCLIC
	// Durchlaufe eine FSM um zwei Shuttles zu verbinden.
	CASE coupleStep OF
		coupleStepWAIT:
			// Warte auf Ready + Befehl.
			IF (trakMove.cmd.test AND trakAsmb.state.ready) THEN
				coupleStep := coupleStepSENDPOS1;
				trakMove.cmd.test := FALSE;
			END_IF;

		coupleStepSENDPOS1:
			// Starte Bewegung des ersten Shuttles.
			FB_move.Sector := ADR(gSecFull);
			FB_move.Position := 0.426;
			FB_move.Axis := ADR(trakAsmb.shuttles[dummyFirst].axis);
			FB_move.Execute := TRUE;
			// Weiter wenn Bewegung abgeschlossen.
			IF FB_move.Done THEN
				FB_move.Execute := FALSE;
				coupleStep := coupleStepSENDPOS2;
			END_IF;

		coupleStepSENDPOS2:
			// Starte Bewegung des zweiten Shuttles.
			FB_move.Sector := ADR(gSecFull);
			FB_move.Position := 0.3;
			FB_move.Axis := ADR(trakAsmb.shuttles[dummySecond].axis);
			FB_move.Execute := TRUE;
			// Weiter wenn Bewegung abgeschlossen.
			IF FB_move.Done THEN
				FB_move.Execute := FALSE;
				coupleStep := coupleStepSETOBJ1;
			END_IF;

		coupleStepSETOBJ1:
			// erstelle ein Convoy
			FB_createConvoy.Axis := ADR(trakAsmb.shuttles[dummyFirst].axis);
			FB_createConvoy.Execute := TRUE;
			// Weiter wenn Convoy erstellt wurde
			IF FB_createConvoy.Done THEN
				FB_createConvoy.Execute := FALSE;
				coupleStep := coupleStepSETOBJ2;
			END_IF;
			// DEBUG: Skip
			//coupleStep := coupleStepCOUPLE;
			// MANUAL

		coupleStepSETOBJ2:
			// TEST
			FB_read1.Axis := ADR(trakAsmb.shuttles[dummyFirst].axis);
			FB_read2.Axis := ADR(trakAsmb.shuttles[dummySecond].axis);
			FB_read1.Enable := TRUE;
			FB_read2.Enable := TRUE;
			// New
			FB_add2Convoy.Parameters.ReferenceShuttle := ADR(trakAsmb.shuttles[dummyFirst].axis);
			FB_add2Convoy.Axis := ADR(trakAsmb.shuttles[dummySecond].axis);
			FB_add2Convoy.Execute := TRUE;
			// OLD
			// Kopplungsobjekt an erstes Shuttle hängen
			//FB_couple.Axis := ADR(trakAsmb.shuttles[dummySecond].axis);
			//FB_couple.CouplingObjectName := 'couplingLoad';
			//FB_couple.Execute := TRUE;
			// Weiter wenn an Objekt angeschlossen.
			IF FB_add2Convoy.Done THEN
				FB_add2Convoy.Execute := FALSE;
				coupleStep := coupleStepDONE;
			END_IF;

		coupleStepCOUPLE:
			// Achsen synchronisieren bez. tatsächlich Koppeln.
			FB_gearin.Master := ADR(trakAsmb.shuttles[dummyFirst].axis);
			FB_gearin.Slave := ADR(trakAsmb.shuttles[dummySecond].axis);
			FB_gearin.Execute := TRUE;
			// Wenn Kopplung aktiv ist, dann sind wir fertig.
			IF FB_gearin.Active THEN
				coupleStep := coupleStepDONE;
			END_IF;

		coupleStepDONE:
			// Master Shuttle bewegen.
			FB_moveCyc.Axis := ADR(trakAsmb.shuttles[dummyFirst].axis);
			FB_moveCyc.Enable := TRUE;
			// Weiter wenn Bewegung abgeschlossen.
			//IF FB_moveCyc.Done THEN
			//	FB_moveAdd.Execute := FALSE;
			//	coupleStep := coupleStepWAIT;
			//END_IF;

	END_CASE;

	// Rufe alle FBs zyklisch auf, werden aber nur berechnet wenn "Enable" oder "Execute" aktiv.
	FB_move();
	FB_couple();
	FB_gearin();
	FB_moveVel();
	FB_moveCyc();
	FB_createConvoy();
	FB_add2Convoy();
	FB_read1();
	FB_read2();

	distance := FB_read1.CyclicPosition - FB_read2.CyclicPosition;

	// Enable der FBs deaktivieren wenn Busy Signal geht oder Fehler ansteht.
	//IF EDGENEG(FB_move.Busy) OR FB_move.Error THEN
	//	FB_move.Execute := FALSE;
	//END_IF;
	//IF EDGENEG(FB_couple.Busy) OR FB_couple.Error THEN
	//	FB_couple.Execute := FALSE;
	//END_IF;

	// Sobald Fehler in GearIn (keine Sanchronisation mehr) auftritt, dann stoppe komplettes Assembly
	IF FB_gearin.Error THEN
		trakAsmb.cmd.power := FALSE;
	END_IF;

END_PROGRAM

PROGRAM _EXIT
	(* Insert code here *)

END_PROGRAM
```

Listed in the project but not available here: Logical/TrakControl/trakMES
